KUKA KRL program: EPS_2_251806_MH50A_A_20260212042250.src

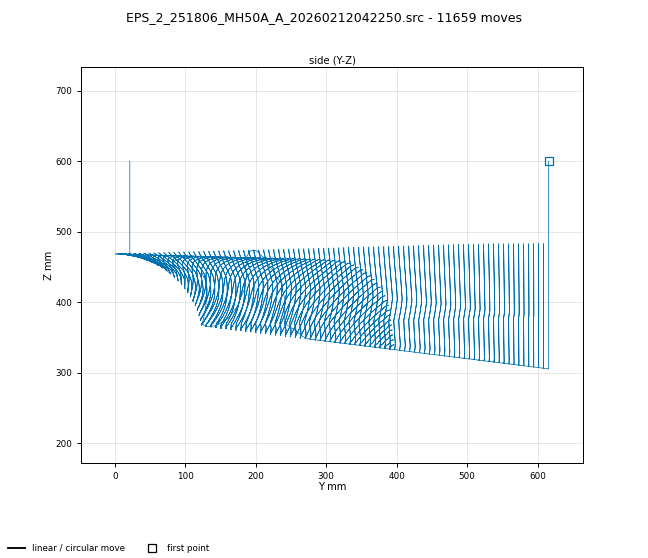
[picture p0: tool path of EPS_2_251806_MH50A_A_20260212042250.src, 11659 of 11661 moves have a stored position in this frame; points joined in program order, loops and branches not executed]
&ACCESS RVP
&REL 4
&COMMENT QRS 19112012
&PARAM EDITMASK = *
DEF PART()
EXT BAS (BAS_COMMAND :IN,REAL :IN )
INT I
BAS (#INITMOV,0 )

;KUKA QRS Post kuka4.cps  Date:22-06-2017 !

File_ID=3022

QRS_PRE_INIT()

;Init var - Until changes are made in qrs_pre_init
Outlet_Square_prg=0
Inlet_1_Square_prg=0
Inlet_2_Square_prg=0
Inlet_3_Square_prg=0
Inlet_4_Square_prg=0
Inlet_5_Square_prg=0

Outlet_1={X 0.000, Y 526.370, Z 382.500, B 0.000, E1 0.000 }
Inlet_1={X 0.000, Y 554.650, Z 357.500, B 0.000, E1 180.000 }
Outlet_1_type=201
Inlet_1_type=0
;QRS#1=Sidecore dimensions
;QRS#2=200-8" PVC SDR 35
;QRS#3=DeadEnd 201
;QRS#4=
;QRS#5=
;QRS#6=
;QRS#7=
;QRS#8=
;QRS#9=12-08 PSX
;QRS#10=

;QRS#11=
;QRS#12=
;QRS#13=
;QRS#14=
;QRS#15=
;QRS#16=1220x127x762 2,5'
;QRS#17=EPS Height
;QRS#18=483
;QRS#19=*
;QRS#20= UPDATED VERSION 22-06-2017
;QRS#21=*
Outlet_Square=0100
Inlet_1_Square=00
Inlet_2_Square=0
Inlet_3_Square=0
Inlet_4_Square=0
Inlet_5_Square=0
Mill_Square=1
Outlet_Square_Prg=204
Inlet_1_Square_prg=0

QRS_INIT()

$ADVANCE=5

; T1
PTP {E1 173.619,E2 173.619}
PTP {X 0,Y 615.481,A -85,B 0,C 180,E1 173.619,E2 173.619,E3 0,E4 0,E5 0,E6 0}
QRS_SPEED_INIT()
LIN {X 0,Y 615.481,Z 600,A -85,B 0,C 180,E1 173.619,E2 173.619,E3 0,E4 0,E5 0,E6 0} C_VEL
LIN {X 0,Y 615.481,Z 315.368,A -85,B 0,C 180,E1 173.619,E2 173.619} C_VEL
LIN {X 0,Y 615.481,Z 307.193,A -85,B 0,C 180,E1 173.619,E2 173.619} C_VEL
LIN {X 0,Y 615.471,Z 305.193,A -85,B 0,C 180,E1 173.433,E2 173.433} C_VEL
LIN {X 0,Y 615.484,Z 305.195,A -85,B 0,C 180,E1 170.802,E2 170.802} C_VEL
LIN {X 0,Y 615.484,Z 305.183,A -85,B 0,C 180,E1 168.14,E2 168.14} C_VEL
LIN {X 0,Y 615.479,Z 305.195,A -85,B 0,C 180,E1 165.451,E2 165.451} C_VEL
LIN {X 0,Y 615.484,Z 305.188,A -85,B 0,C 180,E1 162.73,E2 162.73} C_VEL
LIN {X 0,Y 615.472,Z 305.189,A -85,B 0,C 180,E1 159.967,E2 159.967} C_VEL
LIN {X 0,Y 615.478,Z 305.195,A -85,B 0,C 180,E1 157.656,E2 157.656} C_VEL
LIN {X 0,Y 615.483,Z 305.191,A -85,B 0,C 180,E1 155.009,E2 155.009} C_VEL
LIN {X 0,Y 615.486,Z 305.186,A -85,B 0,C 180,E1 152.823,E2 152.823} C_VEL
LIN {X 0,Y 615.473,Z 305.188,A -85,B 0,C 180,E1 150.207,E2 150.207} C_VEL
LIN {X 0,Y 615.495,Z 305.199,A -85,B 0,C 180,E1 147.544,E2 147.544} C_VEL
LIN {X 0,Y 615.482,Z 305.189,A -85,B 0,C 180,E1 145.185,E2 145.185} C_VEL
LIN {X 0,Y 615.492,Z 305.182,A -85,B 0,C 180,E1 142.759,E2 142.759} C_VEL
LIN {X 0,Y 615.49,Z 305.198,A -85,B 0,C 180,E1 139.91,E2 139.91} C_VEL
LIN {X 0,Y 615.488,Z 305.183,A -85,B 0,C 180,E1 136.952,E2 136.952} C_VEL
LIN {X 0,Y 615.483,Z 305.196,A -85,B 0,C 180,E1 134.15,E2 134.15} C_VEL
LIN {X 0,Y 615.482,Z 305.189,A -85,B 0,C 180,E1 131.474,E2 131.474} C_VEL
LIN {X 0,Y 615.483,Z 305.184,A -85,B 0,C 180,E1 128.904,E2 128.904} C_VEL
LIN {X 0,Y 615.479,Z 305.194,A -85,B 0,C 180,E1 126.425,E2 126.425} C_VEL
LIN {X 0,Y 615.484,Z 305.186,A -85,B 0,C 180,E1 123.534,E2 123.534} C_VEL
LIN {X 0,Y 615.477,Z 305.187,A -85,B 0,C 180,E1 120.92,E2 120.92} C_VEL
LIN {X 0,Y 615.489,Z 305.197,A -85,B 0,C 180,E1 118.451,E2 118.451} C_VEL
LIN {X 0,Y 615.486,Z 305.184,A -85,B 0,C 180,E1 115.57,E2 115.57} C_VEL
LIN {X 0,Y 615.475,Z 305.193,A -85,B 0,C 180,E1 112.845,E2 112.845} C_VEL
LIN {X 0,Y 615.491,Z 305.2,A -85,B 0,C 180,E1 110.559,E2 110.559} C_VEL
LIN {X 0,Y 615.48,Z 305.188,A -85,B 0,C 180,E1 107.957,E2 107.957} C_VEL
LIN {X 0,Y 615.477,Z 305.188,A -85,B 0,C 180,E1 105.226,E2 105.226} C_VEL
LIN {X 0,Y 615.488,Z 305.197,A -85,B 0,C 180,E1 102.53,E2 102.53} C_VEL
LIN {X 0,Y 615.494,Z 305.182,A -85,B 0,C 180,E1 99.862,E2 99.862} C_VEL
LIN {X 0,Y 615.475,Z 305.193,A -85,B 0,C 180,E1 97.216,E2 97.216} C_VEL
LIN {X 0,Y 615.481,Z 305.194,A -85,B 0,C 180,E1 94.585,E2 94.585} C_VEL
LIN {X 0,Y 615.5,Z 305.18,A -85,B 0,C 180,E1 91.963,E2 91.963} C_VEL
LIN {X 0,Y 615.48,Z 305.193,A -85,B 0,C 180,E1 89.346,E2 89.346} C_VEL
LIN {X 0,Y 615.48,Z 305.193,A -85,B 0,C 180,E1 86.727,E2 86.727} C_VEL
LIN {X 0,Y 615.498,Z 305.18,A -85,B 0,C 180,E1 84.102,E2 84.102} C_VEL
LIN {X 0,Y 615.484,Z 305.195,A -85,B 0,C 180,E1 81.463,E2 81.463} C_VEL
LIN {X 0,Y 615.477,Z 305.191,A -85,B 0,C 180,E1 78.807,E2 78.807} C_VEL
LIN {X 0,Y 615.484,Z 305.185,A -85,B 0,C 180,E1 76.067,E2 76.067} C_VEL
LIN {X 0,Y 615.49,Z 305.202,A -85,B 0,C 180,E1 73.414,E2 73.414} C_VEL
LIN {X 0,Y 615.483,Z 305.184,A -85,B 0,C 180,E1 70.662,E2 70.662} C_VEL
LIN {X 0,Y 615.482,Z 305.193,A -85,B 0,C 180,E1 67.863,E2 67.863} C_VEL
LIN {X 0,Y 615.475,Z 305.189,A -85,B 0,C 180,E1 65.008,E2 65.008} C_VEL
LIN {X 0,Y 615.482,Z 305.185,A -85,B 0,C 180,E1 62.823,E2 62.823} C_VEL
LIN {X 0,Y 615.48,Z 305.19,A -85,B 0,C 180,E1 60.206,E2 60.206} C_VEL
LIN {X 0,Y 615.482,Z 305.196,A -85,B 0,C 180,E1 57.542,E2 57.542} C_VEL
LIN {X 0,Y 615.476,Z 305.188,A -85,B 0,C 180,E1 55.184,E2 55.184} C_VEL
LIN {X 0,Y 615.493,Z 305.182,A -85,B 0,C 180,E1 52.758,E2 52.758} C_VEL
LIN {X 0,Y 615.495,Z 305.199,A -85,B 0,C 180,E1 49.91,E2 49.91} C_VEL
LIN {X 0,Y 615.488,Z 305.183,A -85,B 0,C 180,E1 46.952,E2 46.952} C_VEL
LIN {X 0,Y 615.49,Z 305.198,A -85,B 0,C 180,E1 43.998,E2 43.998} C_VEL
LIN {X 0,Y 615.487,Z 305.183,A -85,B 0,C 180,E1 41.095,E2 41.095} C_VEL
LIN {X 0,Y 615.485,Z 305.197,A -85,B 0,C 180,E1 38.068,E2 38.068} C_VEL
LIN {X 0,Y 615.471,Z 305.188,A -85,B 0,C 180,E1 35.616,E2 35.616} C_VEL
LIN {X 0,Y 615.487,Z 305.183,A -85,B 0,C 180,E1 33.236,E2 33.236} C_VEL
LIN {X 0,Y 615.483,Z 305.189,A -85,B 0,C 180,E1 30.919,E2 30.919} C_VEL
LIN {X 0,Y 615.493,Z 305.2,A -85,B 0,C 180,E1 28.452,E2 28.452} C_VEL
LIN {X 0,Y 615.484,Z 305.184,A -85,B 0,C 180,E1 25.569,E2 25.569} C_VEL
LIN {X 0,Y 615.484,Z 305.196,A -85,B 0,C 180,E1 22.844,E2 22.844} C_VEL
LIN {X 0,Y 615.483,Z 305.199,A -85,B 0,C 180,E1 20.557,E2 20.557} C_VEL
LIN {X 0,Y 615.475,Z 305.187,A -85,B 0,C 180,E1 17.957,E2 17.957} C_VEL
LIN {X 0,Y 615.482,Z 305.191,A -85,B 0,C 180,E1 15.226,E2 15.226} C_VEL
LIN {X 0,Y 615.475,Z 305.194,A -85,B 0,C 180,E1 12.53,E2 12.53} C_VEL
LIN {X 0,Y 615.492,Z 305.182,A -85,B 0,C 180,E1 9.862,E2 9.862} C_VEL
LIN {X 0,Y 615.488,Z 305.195,A -85,B 0,C 180,E1 7.215,E2 7.215} C_VEL
LIN {X 0,Y 615.471,Z 305.192,A -85,B 0,C 180,E1 4.584,E2 4.584} C_VEL
LIN {X 0,Y 615.5,Z 305.181,A -85,B 0,C 180,E1 1.963,E2 1.963} C_VEL
LIN {X 0,Y 615.491,Z 305.197,A -85,B 0,C 180,E1 -0.655,E2 -0.655} C_VEL
LIN {X 0,Y 615.469,Z 305.191,A -85,B 0,C 180,E1 -3.273,E2 -3.273} C_VEL
LIN {X 0,Y 615.498,Z 305.181,A -85,B 0,C 180,E1 -5.899,E2 -5.899} C_VEL
LIN {X 0,Y 615.494,Z 305.199,A -85,B 0,C 180,E1 -8.537,E2 -8.537} C_VEL
LIN {X 0,Y 615.468,Z 305.19,A -85,B 0,C 180,E1 -11.194,E2 -11.194} C_VEL
LIN {X 0,Y 615.488,Z 305.187,A -85,B 0,C 180,E1 -13.934,E2 -13.934} C_VEL
LIN {X 0,Y 615.481,Z 305.198,A -85,B 0,C 180,E1 -16.587,E2 -16.587} C_VEL
LIN {X 0,Y 615.48,Z 305.184,A -85,B 0,C 180,E1 -19.339,E2 -19.339} C_VEL
LIN {X 0,Y 615.488,Z 305.197,A -85,B 0,C 180,E1 -22.137,E2 -22.137} C_VEL
LIN {X 0,Y 615.469,Z 305.188,A -85,B 0,C 180,E1 -24.993,E2 -24.993} C_VEL
LIN {X 0,Y 615.489,Z 305.194,A -85,B 0,C 180,E1 -27.915,E2 -27.915} C_VEL
LIN {X 0,Y 615.491,Z 305.2,A -85,B 0,C 180,E1 -30.16,E2 -30.16} C_VEL
LIN {X 0,Y 615.469,Z 305.194,A -85,B 0,C 180,E1 -32.459,E2 -32.459} C_VEL
LIN {X 0,Y 615.47,Z 305.187,A -85,B 0,C 180,E1 -34.817,E2 -34.817} C_VEL
LIN {X 0,Y 615.494,Z 305.183,A -85,B 0,C 180,E1 -37.242,E2 -37.242} C_VEL
LIN {X 0,Y 615.479,Z 305.197,A -85,B 0,C 180,E1 -40.088,E2 -40.088} C_VEL
LIN {X 0,Y 615.465,Z 305.192,A -85,B 0,C 180,E1 -42.355,E2 -42.355} C_VEL
LIN {X 0,Y 615.491,Z 305.184,A -85,B 0,C 180,E1 -45.069,E2 -45.069} C_VEL
LIN {X 0,Y 615.488,Z 305.184,A -85,B 0,C 180,E1 -46.953,E2 -46.953} C_VEL
LIN {X 0,Y 615.499,Z 305.472,A -85,B 0,C 180,E1 -47.648,E2 -47.648} C_VEL
LIN {X 0,Y 615.458,Z 310.077,A -85,B 0,C 180,E1 -50.248,E2 -50.248} C_VEL
LIN {X 0,Y 615.486,Z 315.447,A -85,B 0,C 180,E1 -53.064,E2 -53.064} C_VEL
LIN {X 0,Y 615.483,Z 319.999,A -85,B 0,C 180,E1 -55.3,E2 -55.3} C_VEL
LIN {X 0,Y 615.457,Z 325.099,A -85,B 0,C 180,E1 -57.674,E2 -57.674} C_VEL
LIN {X 0,Y 615.477,Z 330.882,A -85,B 0,C 180,E1 -60.208,E2 -60.208} C_VEL
LIN {X 0,Y 615.484,Z 337.498,A -85,B 0,C 180,E1 -62.956,E2 -62.956} C_VEL
LIN {X 0,Y 615.466,Z 344.318,A -85,B 0,C 180,E1 -65.727,E2 -65.727} C_VEL
LIN {X 0,Y 615.496,Z 351.474,A -85,B 0,C 180,E1 -68.569,E2 -68.569} C_VEL
LIN {X 0,Y 615.462,Z 358.741,A -85,B 0,C 180,E1 -71.403,E2 -71.403} C_VEL
LIN {X 0,Y 615.472,Z 365.762,A -85,B 0,C 180,E1 -74.094,E2 -74.094} C_VEL
LIN {X 0,Y 615.482,Z 372.89,A -85,B 0,C 180,E1 -76.799,E2 -76.799} C_VEL
LIN {X 0,Y 615.496,Z 377.073,A -85,B 0,C 180,E1 -78.369,E2 -78.369} C_VEL
LIN {X 0,Y 615.477,Z 392.864,A -85,B 0,C 180,E1 -78.723,E2 -78.723} C_VEL
LIN {X 0,Y 615.442,Z 405.251,A -85,B 0,C 180,E1 -79.135,E2 -79.135} C_VEL
LIN {X 0,Y 615.442,Z 416.485,A -85,B 0,C 180,E1 -79.639,E2 -79.639} C_VEL
LIN {X 0,Y 615.493,Z 427.995,A -85,B 0,C 180,E1 -80.304,E2 -80.304} C_VEL
LIN {X 0,Y 615.499,Z 438.341,A -85,B 0,C 180,E1 -81.05,E2 -81.05} C_VEL
LIN {X 0,Y 615.497,Z 446.812,A -85,B 0,C 180,E1 -81.794,E2 -81.794} C_VEL
LIN {X 0,Y 615.498,Z 454.606,A -85,B 0,C 180,E1 -82.62,E2 -82.62} C_VEL
LIN {X 0,Y 615.496,Z 462.203,A -85,B 0,C 180,E1 -83.608,E2 -83.608} C_VEL
LIN {X 0,Y 615.498,Z 469.205,A -85,B 0,C 180,E1 -84.759,E2 -84.759} C_VEL
LIN {X 0,Y 615.494,Z 473.851,A -85,B 0,C 180,E1 -85.744,E2 -85.744} C_VEL
LIN {X 0,Y 615.494,Z 477.399,A -85,B 0,C 180,E1 -86.727,E2 -86.727} C_VEL
LIN {X 0,Y 615.497,Z 479.233,A -85,B 0,C 180,E1 -87.382,E2 -87.382} C_VEL
LIN {X 0,Y 615.5,Z 480.607,A -85,B 0,C 180,E1 -88.037,E2 -88.037} C_VEL
LIN {X 0,Y 615.496,Z 482.173,A -85,B 0,C 180,E1 -89.346,E2 -89.346} C_VEL
LIN {X 0,Y 615.494,Z 482.389,A -85,B 0,C 180,E1 -90,E2 -90} C_VEL
LIN {X 0,Y 615.495,Z 481.58,A -85,B 0,C 180,E1 -91.309,E2 -91.309} C_VEL
LIN {X 0,Y 615.5,Z 480.607,A -85,B 0,C 180,E1 -91.963,E2 -91.963} C_VEL
LIN {X 0,Y 615.497,Z 479.233,A -85,B 0,C 180,E1 -92.618,E2 -92.618} C_VEL
LIN {X 0,Y 615.496,Z 476.349,A -85,B 0,C 180,E1 -93.601,E2 -93.601} C_VEL
LIN {X 0,Y 615.498,Z 472.441,A -85,B 0,C 180,E1 -94.584,E2 -94.584} C_VEL
LIN {X 0,Y 615.499,Z 467.405,A -85,B 0,C 180,E1 -95.57,E2 -95.57} C_VEL
LIN {X 0,Y 615.497,Z 460.87,A -85,B 0,C 180,E1 -96.583,E2 -96.583} C_VEL
LIN {X 0,Y 615.497,Z 453.133,A -85,B 0,C 180,E1 -97.545,E2 -97.545} C_VEL
LIN {X 0,Y 615.498,Z 445.045,A -85,B 0,C 180,E1 -98.371,E2 -98.371} C_VEL
LIN {X 0,Y 615.499,Z 435.168,A -85,B 0,C 180,E1 -99.199,E2 -99.199} C_VEL
LIN {X 0,Y 615.478,Z 423.984,A -85,B 0,C 180,E1 -99.945,E2 -99.945} C_VEL
LIN {X 0,Y 615.436,Z 413.032,A -85,B 0,C 180,E1 -100.528,E2 -100.528} C_VEL
LIN {X 0,Y 615.452,Z 400.823,A -85,B 0,C 180,E1 -101.029,E2 -101.029} C_VEL
LIN {X 0,Y 615.49,Z 388.067,A -85,B 0,C 180,E1 -101.401,E2 -101.401} C_VEL
LIN {X 0,Y 615.496,Z 377.073,A -85,B 0,C 180,E1 -101.631,E2 -101.631} C_VEL
LIN {X 0,Y 615.472,Z 370.983,A -85,B 0,C 180,E1 -103.926,E2 -103.926} C_VEL
LIN {X 0,Y 615.454,Z 363.97,A -85,B 0,C 180,E1 -106.587,E2 -106.587} C_VEL
LIN {X 0,Y 615.493,Z 356.829,A -85,B 0,C 180,E1 -109.338,E2 -109.338} C_VEL
LIN {X 0,Y 615.463,Z 349.681,A -85,B 0,C 180,E1 -112.137,E2 -112.137} C_VEL
LIN {X 0,Y 615.487,Z 342.534,A -85,B 0,C 180,E1 -114.992,E2 -114.992} C_VEL
LIN {X 0,Y 615.486,Z 337.172,A -85,B 0,C 180,E1 -117.177,E2 -117.177} C_VEL
LIN {X 0,Y 615.477,Z 330.882,A -85,B 0,C 180,E1 -119.792,E2 -119.792} C_VEL
LIN {X 0,Y 615.457,Z 325.099,A -85,B 0,C 180,E1 -122.326,E2 -122.326} C_VEL
LIN {X 0,Y 615.496,Z 319.757,A -85,B 0,C 180,E1 -124.814,E2 -124.814} C_VEL
LIN {X 0,Y 615.495,Z 314.843,A -85,B 0,C 180,E1 -127.241,E2 -127.241} C_VEL
LIN {X 0,Y 615.458,Z 310.077,A -85,B 0,C 180,E1 -129.752,E2 -129.752} C_VEL
LIN {X 0,Y 615.499,Z 305.472,A -85,B 0,C 180,E1 -132.352,E2 -132.352} C_VEL
LIN {X 0,Y 615.486,Z 305.198,A -85,B 0,C 180,E1 -134.149,E2 -134.149} C_VEL
LIN {X 0,Y 615.488,Z 305.184,A -85,B 0,C 180,E1 -136.952,E2 -136.952} C_VEL
LIN {X 0,Y 615.467,Z 305.189,A -85,B 0,C 180,E1 -139.392,E2 -139.392} C_VEL
LIN {X 0,Y 615.48,Z 305.2,A -85,B 0,C 180,E1 -141.989,E2 -141.989} C_VEL
LIN {X 0,Y 615.484,Z 305.192,A -85,B 0,C 180,E1 -144.384,E2 -144.384} C_VEL
LIN {X 0,Y 615.487,Z 305.184,A -85,B 0,C 180,E1 -146.763,E2 -146.763} C_VEL
LIN {X 0,Y 615.47,Z 305.187,A -85,B 0,C 180,E1 -149.079,E2 -149.079} C_VEL
LIN {X 0,Y 615.474,Z 305.195,A -85,B 0,C 180,E1 -151.552,E2 -151.552} C_VEL
LIN {X 0,Y 615.488,Z 305.185,A -85,B 0,C 180,E1 -154.431,E2 -154.431} C_VEL
LIN {X 0,Y 615.467,Z 305.191,A -85,B 0,C 180,E1 -157.154,E2 -157.154} C_VEL
LIN {X 0,Y 615.48,Z 305.196,A -85,B 0,C 180,E1 -159.444,E2 -159.444} C_VEL
LIN {X 0,Y 615.486,Z 305.19,A -85,B 0,C 180,E1 -162.043,E2 -162.043} C_VEL
LIN {X 0,Y 615.47,Z 305.188,A -85,B 0,C 180,E1 -164.773,E2 -164.773} C_VEL
LIN {X 0,Y 615.487,Z 305.203,A -85,B 0,C 180,E1 -167.47,E2 -167.47} C_VEL
LIN {X 0,Y 615.495,Z 305.183,A -85,B 0,C 180,E1 -170.138,E2 -170.138} C_VEL
LIN {X 0,Y 615.469,Z 305.191,A -85,B 0,C 180,E1 -172.784,E2 -172.784} C_VEL
LIN {X 0,Y 615.492,Z 305.197,A -85,B 0,C 180,E1 -175.415,E2 -175.415} C_VEL
LIN {X 0,Y 615.5,Z 305.181,A -85,B 0,C 180,E1 -178.037,E2 -178.037} C_VEL
LIN {X 0,Y 615.47,Z 305.192,A -85,B 0,C 180,E1 -180.654,E2 -180.654} C_VEL
LIN {X 0,Y 615.49,Z 305.196,A -85,B 0,C 180,E1 -183.273,E2 -183.273} C_VEL
LIN {X 0,Y 615.497,Z 305.181,A -85,B 0,C 180,E1 -185.898,E2 -185.898} C_VEL
LIN {X 0,Y 615.471,Z 305.193,A -85,B 0,C 180,E1 -186.567,E2 -186.567} C_VEL
LIN {X 0,Y 614.806,Z 305.344,A -85,B 0,C 180,E1 -187.113,E2 -187.113} C_VEL
LIN {X 0,Y 611.977,Z 305.748,A -85,B 0,C 180,E1 -187.999,E2 -187.999} C_VEL
LIN {X 0,Y 609.585,Z 306.062,A -85,B 0,C 180,E1 -188.712,E2 -188.712} C_VEL
LIN {X 0,Y 608.549,Z 306.181,A -85,B 0,C 180,E1 -189.262,E2 -189.262} C_VEL
LIN {X 0,Y 608.46,Z 306.189,A -85,B 0,C 180,E1 -189.448,E2 -189.448} C_VEL
LIN {X 0,Y 608.458,Z 306.187,A -85,B 0,C 180,E1 -191.999,E2 -191.999} C_VEL
LIN {X 0,Y 608.469,Z 306.194,A -85,B 0,C 180,E1 -194.72,E2 -194.72} C_VEL
LIN {X 0,Y 608.448,Z 306.189,A -85,B 0,C 180,E1 -197.476,E2 -197.476} C_VEL
LIN {X 0,Y 608.454,Z 306.191,A -85,B 0,C 180,E1 -200.274,E2 -200.274} C_VEL
LIN {X 0,Y 608.456,Z 306.195,A -85,B 0,C 180,E1 -202.476,E2 -202.476} C_VEL
LIN {X 0,Y 608.45,Z 306.189,A -85,B 0,C 180,E1 -205.301,E2 -205.301} C_VEL
LIN {X 0,Y 608.444,Z 306.189,A -85,B 0,C 180,E1 -207.518,E2 -207.518} C_VEL
LIN {X 0,Y 608.456,Z 306.19,A -85,B 0,C 180,E1 -209.97,E2 -209.97} C_VEL
LIN {X 0,Y 608.468,Z 306.194,A -85,B 0,C 180,E1 -212.524,E2 -212.524} C_VEL
LIN {X 0,Y 608.435,Z 306.19,A -85,B 0,C 180,E1 -215.278,E2 -215.278} C_VEL
LIN {X 0,Y 608.468,Z 306.188,A -85,B 0,C 180,E1 -217.746,E2 -217.746} C_VEL
LIN {X 0,Y 608.452,Z 306.196,A -85,B 0,C 180,E1 -220.329,E2 -220.329} C_VEL
LIN {X 0,Y 608.454,Z 306.188,A -85,B 0,C 180,E1 -222.959,E2 -222.959} C_VEL
LIN {X 0,Y 608.454,Z 306.192,A -85,B 0,C 180,E1 -225.736,E2 -225.736} C_VEL
LIN {X 0,Y 608.46,Z 306.188,A -85,B 0,C 180,E1 -228.657,E2 -228.657} C_VEL
LIN {X 0,Y 608.467,Z 306.188,A -85,B 0,C 180,E1 -231.412,E2 -231.412} C_VEL
LIN {X 0,Y 608.473,Z 306.194,A -85,B 0,C 180,E1 -233.95,E2 -233.95} C_VEL
LIN {X 0,Y 608.463,Z 306.189,A -85,B 0,C 180,E1 -236.329,E2 -236.329} C_VEL
LIN {X 0,Y 608.474,Z 306.185,A -85,B 0,C 180,E1 -238.727,E2 -238.727} C_VEL
LIN {X 0,Y 608.47,Z 306.19,A -85,B 0,C 180,E1 -241.38,E2 -241.38} C_VEL
LIN {X 0,Y 608.469,Z 306.187,A -85,B 0,C 180,E1 -244.279,E2 -244.279} C_VEL
LIN {X 0,Y 608.445,Z 306.19,A -85,B 0,C 180,E1 -246.876,E2 -246.876} C_VEL
LIN {X 0,Y 608.467,Z 306.193,A -85,B 0,C 180,E1 -249.32,E2 -249.32} C_VEL
LIN {X 0,Y 608.448,Z 306.192,A -85,B 0,C 180,E1 -251.828,E2 -251.828} C_VEL
LIN {X 0,Y 608.464,Z 306.187,A -85,B 0,C 180,E1 -254.594,E2 -254.594} C_VEL
LIN {X 0,Y 608.474,Z 306.195,A -85,B 0,C 180,E1 -257.323,E2 -257.323} C_VEL
LIN {X 0,Y 608.461,Z 306.187,A -85,B 0,C 180,E1 -260.023,E2 -260.023} C_VEL
LIN {X 0,Y 608.456,Z 306.19,A -85,B 0,C 180,E1 -262.701,E2 -262.701} C_VEL
LIN {X 0,Y 608.46,Z 306.19,A -85,B 0,C 180,E1 -264.698,E2 -264.698} C_VEL
LIN {X 0,Y 608.472,Z 306.191,A -85,B 0,C 180,E1 -267.352,E2 -267.352} C_VEL
LIN {X 0,Y 608.477,Z 306.185,A -85,B 0,C 180,E1 -270,E2 -270} C_VEL
LIN {X 0,Y 608.472,Z 306.191,A -85,B 0,C 180,E1 -272.648,E2 -272.648} C_VEL
LIN {X 0,Y 608.46,Z 306.19,A -85,B 0,C 180,E1 -275.302,E2 -275.302} C_VEL
LIN {X 0,Y 608.477,Z 306.185,A -85,B 0,C 180,E1 -277.967,E2 -277.967} C_VEL
LIN {X 0,Y 608.468,Z 306.192,A -85,B 0,C 180,E1 -280.958,E2 -280.958} C_VEL
LIN {X 0,Y 608.457,Z 306.188,A -85,B 0,C 180,E1 -283.357,E2 -283.357} C_VEL
LIN {X 0,Y 608.458,Z 306.189,A -85,B 0,C 180,E1 -286.094,E2 -286.094} C_VEL
LIN {X 0,Y 608.457,Z 306.192,A -85,B 0,C 180,E1 -288.869,E2 -288.869} C_VEL
LIN {X 0,Y 608.47,Z 306.186,A -85,B 0,C 180,E1 -291.691,E2 -291.691} C_VEL
LIN {X 0,Y 608.45,Z 306.195,A -85,B 0,C 180,E1 -294.571,E2 -294.571} C_VEL
LIN {X 0,Y 608.474,Z 306.185,A -85,B 0,C 180,E1 -297.207,E2 -297.207} C_VEL
LIN {X 0,Y 608.465,Z 306.191,A -85,B 0,C 180,E1 -299.972,E2 -299.972} C_VEL
LIN {X 0,Y 608.458,Z 306.192,A -85,B 0,C 180,E1 -302.523,E2 -302.523} C_VEL
LIN {X 0,Y 608.436,Z 306.19,A -85,B 0,C 180,E1 -305.278,E2 -305.278} C_VEL
LIN {X 0,Y 608.471,Z 306.19,A -85,B 0,C 180,E1 -307.746,E2 -307.746} C_VEL
LIN {X 0,Y 608.45,Z 306.193,A -85,B 0,C 180,E1 -310.33,E2 -310.33} C_VEL
LIN {X 0,Y 608.453,Z 306.187,A -85,B 0,C 180,E1 -312.96,E2 -312.96} C_VEL
LIN {X 0,Y 608.464,Z 306.194,A -85,B 0,C 180,E1 -315.735,E2 -315.735} C_VEL
LIN {X 0,Y 608.457,Z 306.187,A -85,B 0,C 180,E1 -318.658,E2 -318.658} C_VEL
LIN {X 0,Y 608.468,Z 306.19,A -85,B 0,C 180,E1 -321.413,E2 -321.413} C_VEL
LIN {X 0,Y 608.442,Z 306.195,A -85,B 0,C 180,E1 -323.955,E2 -323.955} C_VEL
LIN {X 0,Y 608.446,Z 306.189,A -85,B 0,C 180,E1 -326.329,E2 -326.329} C_VEL
LIN {X 0,Y 608.475,Z 306.185,A -85,B 0,C 180,E1 -328.728,E2 -328.728} C_VEL
LIN {X 0,Y 608.475,Z 306.193,A -85,B 0,C 180,E1 -331.379,E2 -331.379} C_VEL
LIN {X 0,Y 608.441,Z 306.191,A -85,B 0,C 180,E1 -333.965,E2 -333.965} C_VEL
LIN {X 0,Y 608.457,Z 306.188,A -85,B 0,C 180,E1 -336.155,E2 -336.155} C_VEL
LIN {X 0,Y 608.468,Z 306.186,A -85,B 0,C 180,E1 -338.309,E2 -338.309} C_VEL
LIN {X 0,Y 608.469,Z 306.196,A -85,B 0,C 180,E1 -341.284,E2 -341.284} C_VEL
LIN {X 0,Y 608.453,Z 306.188,A -85,B 0,C 180,E1 -343.906,E2 -343.906} C_VEL
LIN {X 0,Y 608.462,Z 306.189,A -85,B 0,C 180,E1 -346.644,E2 -346.644} C_VEL
LIN {X 0,Y 608.457,Z 306.193,A -85,B 0,C 180,E1 -349.35,E2 -349.35} C_VEL
LIN {X 0,Y 608.475,Z 306.185,A -85,B 0,C 180,E1 -352.033,E2 -352.033} C_VEL
LIN {X 0,Y 608.468,Z 306.192,A -85,B 0,C 180,E1 -354.699,E2 -354.699} C_VEL
LIN {X 0,Y 608.463,Z 306.189,A -85,B 0,C 180,E1 -357.352,E2 -357.352} C_VEL
LIN {X 0,Y 608.477,Z 306.185,A -85,B 0,C 180,E1 -360,E2 -360} C_VEL
LIN {X 0,Y 608.478,Z 306.193,A -85,B 0,C 180,E1 -362.648,E2 -362.648} C_VEL
LIN {X 0,Y 608.451,Z 306.189,A -85,B 0,C 180,E1 -365.302,E2 -365.302} C_VEL
LIN {X 0,Y 608.479,Z 306.185,A -85,B 0,C 180,E1 -367.967,E2 -367.967} C_VEL
LIN {X 0,Y 608.463,Z 306.19,A -85,B 0,C 180,E1 -370.954,E2 -370.954} C_VEL
LIN {X 0,Y 608.452,Z 306.188,A -85,B 0,C 180,E1 -373.357,E2 -373.357} C_VEL
LIN {X 0,Y 608.463,Z 306.191,A -85,B 0,C 180,E1 -376.094,E2 -376.094} C_VEL
LIN {X 0,Y 608.451,Z 306.19,A -85,B 0,C 180,E1 -378.87,E2 -378.87} C_VEL
LIN {X 0,Y 608.472,Z 306.187,A -85,B 0,C 180,E1 -381.692,E2 -381.692} C_VEL
LIN {X 0,Y 608.448,Z 306.193,A -85,B 0,C 180,E1 -384.572,E2 -384.572} C_VEL
LIN {X 0,Y 608.472,Z 306.185,A -85,B 0,C 180,E1 -387.206,E2 -387.206} C_VEL
LIN {X 0,Y 608.47,Z 306.194,A -85,B 0,C 180,E1 -389.972,E2 -389.972} C_VEL
LIN {X 0,Y 608.452,Z 306.188,A -85,B 0,C 180,E1 -392.88,E2 -392.88} C_VEL
LIN {X 0,Y 608.436,Z 306.191,A -85,B 0,C 180,E1 -395.278,E2 -395.278} C_VEL
LIN {X 0,Y 608.469,Z 306.193,A -85,B 0,C 180,E1 -397.747,E2 -397.747} C_VEL
LIN {X 0,Y 608.438,Z 306.192,A -85,B 0,C 180,E1 -400.328,E2 -400.328} C_VEL
LIN {X 0,Y 608.478,Z 306.188,A -85,B 0,C 180,E1 -403.31,E2 -403.31} C_VEL
LIN {X 0,Y 608.461,Z 306.191,A -85,B 0,C 180,E1 -406.13,E2 -406.13} C_VEL
LIN {X 0,Y 608.451,Z 306.19,A -85,B 0,C 180,E1 -407.04,E2 -407.04} C_VEL
LIN {X 0,Y 608.491,Z 307.285,A -85,B 0,C 180,E1 -407.941,E2 -407.941} C_VEL
LIN {X 0,Y 608.5,Z 312.161,A -85,B 0,C 180,E1 -410.7,E2 -410.7} C_VEL
LIN {X 0,Y 608.511,Z 316.701,A -85,B 0,C 180,E1 -413.089,E2 -413.089} C_VEL
LIN {X 0,Y 608.458,Z 321.649,A -85,B 0,C 180,E1 -415.53,E2 -415.53} C_VEL
LIN {X 0,Y 608.452,Z 326.723,A -85,B 0,C 180,E1 -417.905,E2 -417.905} C_VEL
LIN {X 0,Y 608.462,Z 331.937,A -85,B 0,C 180,E1 -420.22,E2 -420.22} C_VEL
LIN {X 0,Y 608.459,Z 338.084,A -85,B 0,C 180,E1 -422.797,E2 -422.797} C_VEL
LIN {X 0,Y 608.445,Z 344.512,A -85,B 0,C 180,E1 -425.429,E2 -425.429} C_VEL
LIN {X 0,Y 608.435,Z 349.902,A -85,B 0,C 180,E1 -427.593,E2 -427.593} C_VEL
LIN {X 0,Y 608.448,Z 357.088,A -85,B 0,C 180,E1 -430.429,E2 -430.429} C_VEL
LIN {X 0,Y 608.402,Z 364.274,A -85,B 0,C 180,E1 -433.215,E2 -433.215} C_VEL
LIN {X 0,Y 608.391,Z 369.664,A -85,B 0,C 180,E1 -435.278,E2 -435.278} C_VEL
LIN {X 0,Y 608.449,Z 377.299,A -85,B 0,C 180,E1 -438.169,E2 -438.169} C_VEL
LIN {X 0,Y 608.459,Z 377.616,A -85,B 0,C 180,E1 -438.254,E2 -438.254} C_VEL
LIN {X 0,Y 608.541,Z 390.705,A -85,B 0,C 180,E1 -438.53,E2 -438.53} C_VEL
LIN {X 0,Y 608.472,Z 403.565,A -85,B 0,C 180,E1 -438.941,E2 -438.941} C_VEL
LIN {X 0,Y 608.466,Z 414.924,A -85,B 0,C 180,E1 -439.434,E2 -439.434} C_VEL
LIN {X 0,Y 608.478,Z 425.579,A -85,B 0,C 180,E1 -440.023,E2 -440.023} C_VEL
LIN {X 0,Y 608.483,Z 436.476,A -85,B 0,C 180,E1 -440.778,E2 -440.778} C_VEL
LIN {X 0,Y 608.475,Z 447.114,A -85,B 0,C 180,E1 -441.699,E2 -441.699} C_VEL
LIN {X 0,Y 608.471,Z 454.96,A -85,B 0,C 180,E1 -442.534,E2 -442.534} C_VEL
LIN {X 0,Y 608.461,Z 462.286,A -85,B 0,C 180,E1 -443.485,E2 -443.485} C_VEL
LIN {X 0,Y 608.451,Z 467.865,A -85,B 0,C 180,E1 -444.366,E2 -444.366} C_VEL
LIN {X 0,Y 608.432,Z 472.95,A -85,B 0,C 180,E1 -445.362,E2 -445.362} C_VEL
LIN {X 0,Y 608.449,Z 476.896,A -85,B 0,C 180,E1 -446.358,E2 -446.358} C_VEL
LIN {X 0,Y 608.425,Z 479.808,A -85,B 0,C 180,E1 -447.352,E2 -447.352} C_VEL
LIN {X 0,Y 608.445,Z 481.201,A -85,B 0,C 180,E1 -448.014,E2 -448.014} C_VEL
LIN {X 0,Y 608.438,Z 482.783,A -85,B 0,C 180,E1 -449.338,E2 -449.338} C_VEL
LIN {X 0,Y 608.434,Z 482.998,A -85,B 0,C 180,E1 -450,E2 -450} C_VEL
LIN {X 0,Y 608.448,Z 482.184,A -85,B 0,C 180,E1 -451.324,E2 -451.324} C_VEL
LIN {X 0,Y 608.445,Z 481.201,A -85,B 0,C 180,E1 -451.986,E2 -451.986} C_VEL
LIN {X 0,Y 608.425,Z 479.808,A -85,B 0,C 180,E1 -452.648,E2 -452.648} C_VEL
LIN {X 0,Y 608.449,Z 476.896,A -85,B 0,C 180,E1 -453.642,E2 -453.642} C_VEL
LIN {X 0,Y 608.432,Z 472.95,A -85,B 0,C 180,E1 -454.638,E2 -454.638} C_VEL
LIN {X 0,Y 608.451,Z 467.865,A -85,B 0,C 180,E1 -455.634,E2 -455.634} C_VEL
LIN {X 0,Y 608.442,Z 461.472,A -85,B 0,C 180,E1 -456.633,E2 -456.633} C_VEL
LIN {X 0,Y 608.475,Z 453.479,A -85,B 0,C 180,E1 -457.633,E2 -457.633} C_VEL
LIN {X 0,Y 608.487,Z 445.338,A -85,B 0,C 180,E1 -458.468,E2 -458.468} C_VEL
LIN {X 0,Y 608.487,Z 435.398,A -85,B 0,C 180,E1 -459.306,E2 -459.306} C_VEL
LIN {X 0,Y 608.484,Z 424.168,A -85,B 0,C 180,E1 -460.061,E2 -460.061} C_VEL
LIN {X 0,Y 608.46,Z 411.891,A -85,B 0,C 180,E1 -460.712,E2 -460.712} C_VEL
LIN {X 0,Y 608.487,Z 400.098,A -85,B 0,C 180,E1 -461.186,E2 -461.186} C_VEL
LIN {X 0,Y 608.548,Z 387.262,A -85,B 0,C 180,E1 -461.554,E2 -461.554} C_VEL
LIN {X 0,Y 608.436,Z 377.467,A -85,B 0,C 180,E1 -461.768,E2 -461.768} C_VEL
LIN {X 0,Y 608.426,Z 371.46,A -85,B 0,C 180,E1 -464.038,E2 -464.038} C_VEL
LIN {X 0,Y 608.402,Z 364.274,A -85,B 0,C 180,E1 -466.785,E2 -466.785} C_VEL
LIN {X 0,Y 608.449,Z 357.088,A -85,B 0,C 180,E1 -469.571,E2 -469.571} C_VEL
LIN {X 0,Y 608.431,Z 349.746,A -85,B 0,C 180,E1 -472.469,E2 -472.469} C_VEL
LIN {X 0,Y 608.445,Z 344.512,A -85,B 0,C 180,E1 -474.571,E2 -474.571} C_VEL
LIN {X 0,Y 608.459,Z 338.084,A -85,B 0,C 180,E1 -477.203,E2 -477.203} C_VEL
LIN {X 0,Y 608.462,Z 331.489,A -85,B 0,C 180,E1 -479.97,E2 -479.97} C_VEL
LIN {X 0,Y 608.461,Z 325.787,A -85,B 0,C 180,E1 -482.522,E2 -482.522} C_VEL
LIN {X 0,Y 608.471,Z 319.985,A -85,B 0,C 180,E1 -485.276,E2 -485.276} C_VEL
LIN {X 0,Y 608.487,Z 315.09,A -85,B 0,C 180,E1 -487.745,E2 -487.745} C_VEL
LIN {X 0,Y 608.485,Z 310.293,A -85,B 0,C 180,E1 -490.332,E2 -490.332} C_VEL
LIN {X 0,Y 608.514,Z 306.802,A -85,B 0,C 180,E1 -492.339,E2 -492.339} C_VEL
LIN {X 0,Y 608.451,Z 306.191,A -85,B 0,C 180,E1 -492.96,E2 -492.96} C_VEL
LIN {X 0,Y 608.443,Z 306.192,A -85,B 0,C 180,E1 -495.737,E2 -495.737} C_VEL
LIN {X 0,Y 608.456,Z 306.193,A -85,B 0,C 180,E1 -497.938,E2 -497.938} C_VEL
LIN {X 0,Y 608.48,Z 306.186,A -85,B 0,C 180,E1 -500.701,E2 -500.701} C_VEL
LIN {X 0,Y 608.449,Z 306.188,A -85,B 0,C 180,E1 -503.084,E2 -503.084} C_VEL
LIN {X 0,Y 608.459,Z 306.19,A -85,B 0,C 180,E1 -505.53,E2 -505.53} C_VEL
LIN {X 0,Y 608.46,Z 306.196,A -85,B 0,C 180,E1 -507.905,E2 -507.905} C_VEL
LIN {X 0,Y 608.472,Z 306.19,A -85,B 0,C 180,E1 -510.22,E2 -510.22} C_VEL
LIN {X 0,Y 608.472,Z 306.185,A -85,B 0,C 180,E1 -512.794,E2 -512.794} C_VEL
LIN {X 0,Y 608.448,Z 306.193,A -85,B 0,C 180,E1 -515.428,E2 -515.428} C_VEL
LIN {X 0,Y 608.472,Z 306.187,A -85,B 0,C 180,E1 -518.308,E2 -518.308} C_VEL
LIN {X 0,Y 608.466,Z 306.19,A -85,B 0,C 180,E1 -521.285,E2 -521.285} C_VEL
LIN {X 0,Y 608.463,Z 306.191,A -85,B 0,C 180,E1 -523.906,E2 -523.906} C_VEL
LIN {X 0,Y 608.452,Z 306.188,A -85,B 0,C 180,E1 -526.643,E2 -526.643} C_VEL
LIN {X 0,Y 608.463,Z 306.195,A -85,B 0,C 180,E1 -529.35,E2 -529.35} C_VEL
LIN {X 0,Y 608.479,Z 306.185,A -85,B 0,C 180,E1 -532.033,E2 -532.033} C_VEL
LIN {X 0,Y 608.45,Z 306.189,A -85,B 0,C 180,E1 -534.698,E2 -534.698} C_VEL
LIN {X 0,Y 608.478,Z 306.193,A -85,B 0,C 180,E1 -537.352,E2 -537.352} C_VEL
LIN {X 0,Y 608.477,Z 306.185,A -85,B 0,C 180,E1 -540,E2 -540} C_VEL
LIN {X 0,Y 608.463,Z 306.189,A -85,B 0,C 180,E1 -542.648,E2 -542.648} C_VEL
LIN {X 0,Y 608.468,Z 306.192,A -85,B 0,C 180,E1 -545.301,E2 -545.301} C_VEL
LIN {X 0,Y 608.475,Z 306.185,A -85,B 0,C 180,E1 -547.967,E2 -547.967} C_VEL
LIN {X 0,Y 608.46,Z 306.189,A -85,B 0,C 180,E1 -549.448,E2 -549.448} C_VEL
LIN {X 0,Y 607.781,Z 306.274,A -85,B 0,C 180,E1 -550,E2 -550} C_VEL
LIN {X 0,Y 604.927,Z 306.637,A -85,B 0,C 180,E1 -550.897,E2 -550.897} C_VEL
LIN {X 0,Y 602.522,Z 306.931,A -85,B 0,C 180,E1 -551.619,E2 -551.619} C_VEL
LIN {X 0,Y 601.49,Z 307.056,A -85,B 0,C 180,E1 -552.175,E2 -552.175} C_VEL
LIN {X 0,Y 601.405,Z 307.068,A -85,B 0,C 180,E1 -552.364,E2 -552.364} C_VEL
LIN {X 0,Y 601.425,Z 307.072,A -85,B 0,C 180,E1 -554.897,E2 -554.897} C_VEL
LIN {X 0,Y 601.43,Z 307.069,A -85,B 0,C 180,E1 -556.986,E2 -556.986} C_VEL
LIN {X 0,Y 601.401,Z 307.066,A -85,B 0,C 180,E1 -559.809,E2 -559.809} C_VEL
LIN {X 0,Y 601.413,Z 307.075,A -85,B 0,C 180,E1 -562.605,E2 -562.605} C_VEL
LIN {X 0,Y 601.399,Z 307.071,A -85,B 0,C 180,E1 -564.878,E2 -564.878} C_VEL
LIN {X 0,Y 601.414,Z 307.065,A -85,B 0,C 180,E1 -567.363,E2 -567.363} C_VEL
LIN {X 0,Y 601.424,Z 307.068,A -85,B 0,C 180,E1 -570.148,E2 -570.148} C_VEL
LIN {X 0,Y 601.427,Z 307.068,A -85,B 0,C 180,E1 -572.717,E2 -572.717} C_VEL
LIN {X 0,Y 601.392,Z 307.068,A -85,B 0,C 180,E1 -575.112,E2 -575.112} C_VEL
LIN {X 0,Y 601.433,Z 307.062,A -85,B 0,C 180,E1 -577.419,E2 -577.419} C_VEL
LIN {X 0,Y 601.409,Z 307.072,A -85,B 0,C 180,E1 -579.995,E2 -579.995} C_VEL
LIN {X 0,Y 601.41,Z 307.067,A -85,B 0,C 180,E1 -582.67,E2 -582.67} C_VEL
LIN {X 0,Y 601.422,Z 307.065,A -85,B 0,C 180,E1 -585.482,E2 -585.482} C_VEL
LIN {X 0,Y 601.423,Z 307.067,A -85,B 0,C 180,E1 -588.406,E2 -588.406} C_VEL
LIN {X 0,Y 601.435,Z 307.062,A -85,B 0,C 180,E1 -590.876,E2 -590.876} C_VEL
LIN {X 0,Y 601.439,Z 307.069,A -85,B 0,C 180,E1 -593.734,E2 -593.734} C_VEL
LIN {X 0,Y 601.426,Z 307.063,A -85,B 0,C 180,E1 -596.687,E2 -596.687} C_VEL
LIN {X 0,Y 601.427,Z 307.064,A -85,B 0,C 180,E1 -599.059,E2 -599.059} C_VEL
LIN {X 0,Y 601.43,Z 307.067,A -85,B 0,C 180,E1 -601.373,E2 -601.373} C_VEL
LIN {X 0,Y 601.402,Z 307.077,A -85,B 0,C 180,E1 -603.636,E2 -603.636} C_VEL
LIN {X 0,Y 601.416,Z 307.064,A -85,B 0,C 180,E1 -606.59,E2 -606.59} C_VEL
LIN {X 0,Y 601.43,Z 307.073,A -85,B 0,C 180,E1 -609.478,E2 -609.478} C_VEL
LIN {X 0,Y 601.393,Z 307.067,A -85,B 0,C 180,E1 -612.312,E2 -612.312} C_VEL
LIN {X 0,Y 601.409,Z 307.065,A -85,B 0,C 180,E1 -614.409,E2 -614.409} C_VEL
LIN {X 0,Y 601.418,Z 307.072,A -85,B 0,C 180,E1 -617.172,E2 -617.172} C_VEL
LIN {X 0,Y 601.437,Z 307.063,A -85,B 0,C 180,E1 -619.905,E2 -619.905} C_VEL
LIN {X 0,Y 601.435,Z 307.064,A -85,B 0,C 180,E1 -622.615,E2 -622.615} C_VEL
LIN {X 0,Y 601.418,Z 307.071,A -85,B 0,C 180,E1 -625.308,E2 -625.308} C_VEL
LIN {X 0,Y 601.438,Z 307.062,A -85,B 0,C 180,E1 -627.991,E2 -627.991} C_VEL
LIN {X 0,Y 601.446,Z 307.066,A -85,B 0,C 180,E1 -630.67,E2 -630.67} C_VEL
LIN {X 0,Y 601.425,Z 307.067,A -85,B 0,C 180,E1 -633.35,E2 -633.35} C_VEL
LIN {X 0,Y 601.441,Z 307.062,A -85,B 0,C 180,E1 -636.037,E2 -636.037} C_VEL
LIN {X 0,Y 601.433,Z 307.072,A -85,B 0,C 180,E1 -638.738,E2 -638.738} C_VEL
LIN {X 0,Y 601.431,Z 307.063,A -85,B 0,C 180,E1 -641.458,E2 -641.458} C_VEL
LIN {X 0,Y 601.417,Z 307.068,A -85,B 0,C 180,E1 -644.205,E2 -644.205} C_VEL
LIN {X 0,Y 601.43,Z 307.067,A -85,B 0,C 180,E1 -646.986,E2 -646.986} C_VEL
LIN {X 0,Y 601.404,Z 307.067,A -85,B 0,C 180,E1 -649.809,E2 -649.809} C_VEL
LIN {X 0,Y 601.412,Z 307.072,A -85,B 0,C 180,E1 -652.606,E2 -652.606} C_VEL
LIN {X 0,Y 601.4,Z 307.069,A -85,B 0,C 180,E1 -654.879,E2 -654.879} C_VEL
LIN {X 0,Y 601.419,Z 307.067,A -85,B 0,C 180,E1 -657.867,E2 -657.867} C_VEL
LIN {X 0,Y 601.425,Z 307.072,A -85,B 0,C 180,E1 -660.164,E2 -660.164} C_VEL
LIN {X 0,Y 601.419,Z 307.066,A -85,B 0,C 180,E1 -662.716,E2 -662.716} C_VEL
LIN {X 0,Y 601.391,Z 307.067,A -85,B 0,C 180,E1 -665.112,E2 -665.112} C_VEL
LIN {X 0,Y 601.434,Z 307.063,A -85,B 0,C 180,E1 -667.419,E2 -667.419} C_VEL
LIN {X 0,Y 601.41,Z 307.075,A -85,B 0,C 180,E1 -669.995,E2 -669.995} C_VEL
LIN {X 0,Y 601.408,Z 307.066,A -85,B 0,C 180,E1 -672.67,E2 -672.67} C_VEL
LIN {X 0,Y 601.422,Z 307.067,A -85,B 0,C 180,E1 -675.482,E2 -675.482} C_VEL
LIN {X 0,Y 601.422,Z 307.065,A -85,B 0,C 180,E1 -678.407,E2 -678.407} C_VEL
LIN {X 0,Y 601.435,Z 307.062,A -85,B 0,C 180,E1 -680.876,E2 -680.876} C_VEL
LIN {X 0,Y 601.402,Z 307.071,A -85,B 0,C 180,E1 -683.418,E2 -683.418} C_VEL
LIN {X 0,Y 601.428,Z 307.066,A -85,B 0,C 180,E1 -686.065,E2 -686.065} C_VEL
LIN {X 0,Y 601.438,Z 307.061,A -85,B 0,C 180,E1 -688.542,E2 -688.542} C_VEL
LIN {X 0,Y 601.434,Z 307.07,A -85,B 0,C 180,E1 -691.374,E2 -691.374} C_VEL
LIN {X 0,Y 601.4,Z 307.073,A -85,B 0,C 180,E1 -693.637,E2 -693.637} C_VEL
LIN {X 0,Y 601.416,Z 307.065,A -85,B 0,C 180,E1 -696.59,E2 -696.59} C_VEL
LIN {X 0,Y 601.427,Z 307.07,A -85,B 0,C 180,E1 -699.478,E2 -699.478} C_VEL
LIN {X 0,Y 601.392,Z 307.067,A -85,B 0,C 180,E1 -702.312,E2 -702.312} C_VEL
LIN {X 0,Y 601.409,Z 307.065,A -85,B 0,C 180,E1 -704.409,E2 -704.409} C_VEL
LIN {X 0,Y 601.415,Z 307.074,A -85,B 0,C 180,E1 -707.172,E2 -707.172} C_VEL
LIN {X 0,Y 601.434,Z 307.062,A -85,B 0,C 180,E1 -709.905,E2 -709.905} C_VEL
LIN {X 0,Y 601.441,Z 307.065,A -85,B 0,C 180,E1 -712.615,E2 -712.615} C_VEL
LIN {X 0,Y 601.411,Z 307.069,A -85,B 0,C 180,E1 -715.308,E2 -715.308} C_VEL
LIN {X 0,Y 601.437,Z 307.062,A -85,B 0,C 180,E1 -717.991,E2 -717.991} C_VEL
LIN {X 0,Y 601.455,Z 307.067,A -85,B 0,C 180,E1 -720.67,E2 -720.67} C_VEL
LIN {X 0,Y 601.417,Z 307.066,A -85,B 0,C 180,E1 -723.35,E2 -723.35} C_VEL
LIN {X 0,Y 601.442,Z 307.062,A -85,B 0,C 180,E1 -726.037,E2 -726.037} C_VEL
LIN {X 0,Y 601.437,Z 307.07,A -85,B 0,C 180,E1 -728.738,E2 -728.738} C_VEL
LIN {X 0,Y 601.411,Z 307.065,A -85,B 0,C 180,E1 -731.459,E2 -731.459} C_VEL
LIN {X 0,Y 601.42,Z 307.069,A -85,B 0,C 180,E1 -734.206,E2 -734.206} C_VEL
LIN {X 0,Y 601.419,Z 307.066,A -85,B 0,C 180,E1 -736.987,E2 -736.987} C_VEL
LIN {X 0,Y 601.404,Z 307.068,A -85,B 0,C 180,E1 -739.81,E2 -739.81} C_VEL
LIN {X 0,Y 601.411,Z 307.068,A -85,B 0,C 180,E1 -742.683,E2 -742.683} C_VEL
LIN {X 0,Y 601.398,Z 307.068,A -85,B 0,C 180,E1 -744.879,E2 -744.879} C_VEL
LIN {X 0,Y 601.413,Z 307.065,A -85,B 0,C 180,E1 -747.362,E2 -747.362} C_VEL
LIN {X 0,Y 601.429,Z 307.072,A -85,B 0,C 180,E1 -750.164,E2 -750.164} C_VEL
LIN {X 0,Y 601.413,Z 307.066,A -85,B 0,C 180,E1 -752.714,E2 -752.714} C_VEL
LIN {X 0,Y 601.389,Z 307.068,A -85,B 0,C 180,E1 -755.111,E2 -755.111} C_VEL
LIN {X 0,Y 601.436,Z 307.065,A -85,B 0,C 180,E1 -757.419,E2 -757.419} C_VEL
LIN {X 0,Y 601.413,Z 307.073,A -85,B 0,C 180,E1 -759.995,E2 -759.995} C_VEL
LIN {X 0,Y 601.407,Z 307.066,A -85,B 0,C 180,E1 -762.671,E2 -762.671} C_VEL
LIN {X 0,Y 601.428,Z 307.07,A -85,B 0,C 180,E1 -765.482,E2 -765.482} C_VEL
LIN {X 0,Y 601.429,Z 307.067,A -85,B 0,C 180,E1 -766.428,E2 -766.428} C_VEL
LIN {X 0,Y 601.493,Z 307.667,A -85,B 0,C 180,E1 -767.401,E2 -767.401} C_VEL
LIN {X 0,Y 601.464,Z 312.149,A -85,B 0,C 180,E1 -770.009,E2 -770.009} C_VEL
LIN {X 0,Y 601.509,Z 316.937,A -85,B 0,C 180,E1 -772.609,E2 -772.609} C_VEL
LIN {X 0,Y 601.471,Z 321.813,A -85,B 0,C 180,E1 -775.072,E2 -775.072} C_VEL
LIN {X 0,Y 601.434,Z 326.847,A -85,B 0,C 180,E1 -777.485,E2 -777.485} C_VEL
LIN {X 0,Y 601.43,Z 332.026,A -85,B 0,C 180,E1 -779.852,E2 -779.852} C_VEL
LIN {X 0,Y 601.383,Z 337.326,A -85,B 0,C 180,E1 -782.131,E2 -782.131} C_VEL
LIN {X 0,Y 601.411,Z 342.716,A -85,B 0,C 180,E1 -784.382,E2 -784.382} C_VEL
LIN {X 0,Y 601.372,Z 349.902,A -85,B 0,C 180,E1 -787.316,E2 -787.316} C_VEL
LIN {X 0,Y 601.369,Z 357.088,A -85,B 0,C 180,E1 -790.189,E2 -790.189} C_VEL
LIN {X 0,Y 601.336,Z 364.274,A -85,B 0,C 180,E1 -793.011,E2 -793.011} C_VEL
LIN {X 0,Y 601.335,Z 371.46,A -85,B 0,C 180,E1 -795.793,E2 -795.793} C_VEL
LIN {X 0,Y 601.37,Z 377.579,A -85,B 0,C 180,E1 -798.113,E2 -798.113} C_VEL
LIN {X 0,Y 601.609,Z 387.254,A -85,B 0,C 180,E1 -798.31,E2 -798.31} C_VEL
LIN {X 0,Y 601.531,Z 399.26,A -85,B 0,C 180,E1 -798.656,E2 -798.656} C_VEL
LIN {X 0,Y 601.486,Z 411.437,A -85,B 0,C 180,E1 -799.141,E2 -799.141} C_VEL
LIN {X 0,Y 601.476,Z 422.757,A -85,B 0,C 180,E1 -799.736,E2 -799.736} C_VEL
LIN {X 0,Y 601.462,Z 434.248,A -85,B 0,C 180,E1 -800.5,E2 -800.5} C_VEL
LIN {X 0,Y 601.436,Z 443.521,A -85,B 0,C 180,E1 -801.262,E2 -801.262} C_VEL
LIN {X 0,Y 601.4,Z 451.994,A -85,B 0,C 180,E1 -802.108,E2 -802.108} C_VEL
LIN {X 0,Y 601.382,Z 460.239,A -85,B 0,C 180,E1 -803.12,E2 -803.12} C_VEL
LIN {X 0,Y 601.361,Z 465.868,A -85,B 0,C 180,E1 -803.962,E2 -803.962} C_VEL
LIN {X 0,Y 601.345,Z 471.365,A -85,B 0,C 180,E1 -804.971,E2 -804.971} C_VEL
LIN {X 0,Y 601.347,Z 475.672,A -85,B 0,C 180,E1 -805.979,E2 -805.979} C_VEL
LIN {X 0,Y 601.344,Z 477.959,A -85,B 0,C 180,E1 -806.65,E2 -806.65} C_VEL
LIN {X 0,Y 601.325,Z 479.805,A -85,B 0,C 180,E1 -807.32,E2 -807.32} C_VEL
LIN {X 0,Y 601.343,Z 481.199,A -85,B 0,C 180,E1 -807.991,E2 -807.991} C_VEL
LIN {X 0,Y 601.339,Z 482.783,A -85,B 0,C 180,E1 -809.33,E2 -809.33} C_VEL
LIN {X 0,Y 601.335,Z 482.991,A -85,B 0,C 180,E1 -810,E2 -810} C_VEL
LIN {X 0,Y 601.347,Z 482.185,A -85,B 0,C 180,E1 -811.339,E2 -811.339} C_VEL
LIN {X 0,Y 601.343,Z 481.199,A -85,B 0,C 180,E1 -812.009,E2 -812.009} C_VEL
LIN {X 0,Y 601.325,Z 479.805,A -85,B 0,C 180,E1 -812.68,E2 -812.68} C_VEL
LIN {X 0,Y 601.368,Z 476.894,A -85,B 0,C 180,E1 -813.685,E2 -813.685} C_VEL
LIN {X 0,Y 601.336,Z 472.949,A -85,B 0,C 180,E1 -814.693,E2 -814.693} C_VEL
LIN {X 0,Y 601.374,Z 467.857,A -85,B 0,C 180,E1 -815.701,E2 -815.701} C_VEL
LIN {X 0,Y 601.382,Z 461.47,A -85,B 0,C 180,E1 -816.711,E2 -816.711} C_VEL
LIN {X 0,Y 601.396,Z 453.482,A -85,B 0,C 180,E1 -817.723,E2 -817.723} C_VEL
LIN {X 0,Y 601.423,Z 445.341,A -85,B 0,C 180,E1 -818.568,E2 -818.568} C_VEL
LIN {X 0,Y 601.455,Z 435.386,A -85,B 0,C 180,E1 -819.415,E2 -819.415} C_VEL
LIN {X 0,Y 601.465,Z 425.572,A -85,B 0,C 180,E1 -820.094,E2 -820.094} C_VEL
LIN {X 0,Y 601.474,Z 414.928,A -85,B 0,C 180,E1 -820.69,E2 -820.69} C_VEL
LIN {X 0,Y 601.515,Z 401.857,A -85,B 0,C 180,E1 -821.253,E2 -821.253} C_VEL
LIN {X 0,Y 601.578,Z 389.045,A -85,B 0,C 180,E1 -821.647,E2 -821.647} C_VEL
LIN {X 0,Y 601.456,Z 378.412,A -85,B 0,C 180,E1 -821.872,E2 -821.872} C_VEL
LIN {X 0,Y 601.341,Z 377.467,A -85,B 0,C 180,E1 -821.909,E2 -821.909} C_VEL
LIN {X 0,Y 601.327,Z 369.664,A -85,B 0,C 180,E1 -824.899,E2 -824.899} C_VEL
LIN {X 0,Y 601.368,Z 362.478,A -85,B 0,C 180,E1 -827.689,E2 -827.689} C_VEL
LIN {X 0,Y 601.356,Z 355.291,A -85,B 0,C 180,E1 -830.524,E2 -830.524} C_VEL
LIN {X 0,Y 601.386,Z 348.105,A -85,B 0,C 180,E1 -833.412,E2 -833.412} C_VEL
LIN {X 0,Y 601.396,Z 342.125,A -85,B 0,C 180,E1 -835.863,E2 -835.863} C_VEL
LIN {X 0,Y 601.433,Z 335.151,A -85,B 0,C 180,E1 -838.788,E2 -838.788} C_VEL
LIN {X 0,Y 601.443,Z 329.137,A -85,B 0,C 180,E1 -841.458,E2 -841.458} C_VEL
LIN {X 0,Y 601.456,Z 323.483,A -85,B 0,C 180,E1 -844.116,E2 -844.116} C_VEL
LIN {X 0,Y 601.494,Z 318.523,A -85,B 0,C 180,E1 -846.576,E2 -846.576} C_VEL
LIN {X 0,Y 601.512,Z 313.712,A -85,B 0,C 180,E1 -849.119,E2 -849.119} C_VEL
LIN {X 0,Y 601.511,Z 309.077,A -85,B 0,C 180,E1 -851.757,E2 -851.757} C_VEL
LIN {X 0,Y 601.465,Z 307.554,A -85,B 0,C 180,E1 -852.665,E2 -852.665} C_VEL
LIN {X 0,Y 601.429,Z 307.069,A -85,B 0,C 180,E1 -853.586,E2 -853.586} C_VEL
LIN {X 0,Y 601.431,Z 307.07,A -85,B 0,C 180,E1 -856.427,E2 -856.427} C_VEL
LIN {X 0,Y 601.414,Z 307.065,A -85,B 0,C 180,E1 -859.125,E2 -859.125} C_VEL
LIN {X 0,Y 601.413,Z 307.069,A -85,B 0,C 180,E1 -861.731,E2 -861.731} C_VEL
LIN {X 0,Y 601.387,Z 307.075,A -85,B 0,C 180,E1 -864.245,E2 -864.245} C_VEL
LIN {X 0,Y 601.426,Z 307.064,A -85,B 0,C 180,E1 -866.686,E2 -866.686} C_VEL
LIN {X 0,Y 601.412,Z 307.065,A -85,B 0,C 180,E1 -869.057,E2 -869.057} C_VEL
LIN {X 0,Y 601.421,Z 307.066,A -85,B 0,C 180,E1 -871.372,E2 -871.372} C_VEL
LIN {X 0,Y 601.397,Z 307.074,A -85,B 0,C 180,E1 -873.636,E2 -873.636} C_VEL
LIN {X 0,Y 601.459,Z 307.068,A -85,B 0,C 180,E1 -875.859,E2 -875.859} C_VEL
LIN {X 0,Y 601.406,Z 307.065,A -85,B 0,C 180,E1 -878.76,E2 -878.76} C_VEL
LIN {X 0,Y 601.419,Z 307.074,A -85,B 0,C 180,E1 -881.608,E2 -881.608} C_VEL
LIN {X 0,Y 601.441,Z 307.069,A -85,B 0,C 180,E1 -883.713,E2 -883.713} C_VEL
LIN {X 0,Y 601.41,Z 307.065,A -85,B 0,C 180,E1 -886.484,E2 -886.484} C_VEL
LIN {X 0,Y 601.416,Z 307.071,A -85,B 0,C 180,E1 -889.224,E2 -889.224} C_VEL
LIN {X 0,Y 601.442,Z 307.063,A -85,B 0,C 180,E1 -891.939,E2 -891.939} C_VEL
LIN {X 0,Y 601.419,Z 307.065,A -85,B 0,C 180,E1 -894.635,E2 -894.635} C_VEL
LIN {X 0,Y 601.443,Z 307.07,A -85,B 0,C 180,E1 -897.321,E2 -897.321} C_VEL
LIN {X 0,Y 601.445,Z 307.061,A -85,B 0,C 180,E1 -900,E2 -900} C_VEL
LIN {X 0,Y 601.431,Z 307.066,A -85,B 0,C 180,E1 -902.679,E2 -902.679} C_VEL
LIN {X 0,Y 601.433,Z 307.067,A -85,B 0,C 180,E1 -905.364,E2 -905.364} C_VEL
LIN {X 0,Y 601.437,Z 307.061,A -85,B 0,C 180,E1 -908.06,E2 -908.06} C_VEL
LIN {X 0,Y 601.423,Z 307.072,A -85,B 0,C 180,E1 -911.012,E2 -911.012} C_VEL
LIN {X 0,Y 601.405,Z 307.068,A -85,B 0,C 180,E1 -912.364,E2 -912.364} C_VEL
LIN {X 0,Y 600.738,Z 307.158,A -85,B 0,C 180,E1 -912.923,E2 -912.923} C_VEL
LIN {X 0,Y 597.89,Z 307.515,A -85,B 0,C 180,E1 -913.831,E2 -913.831} C_VEL
LIN {X 0,Y 595.481,Z 307.813,A -85,B 0,C 180,E1 -914.561,E2 -914.561} C_VEL
LIN {X 0,Y 594.443,Z 307.938,A -85,B 0,C 180,E1 -915.125,E2 -915.125} C_VEL
LIN {X 0,Y 594.357,Z 307.946,A -85,B 0,C 180,E1 -915.316,E2 -915.316} C_VEL
LIN {X 0,Y 594.35,Z 307.945,A -85,B 0,C 180,E1 -917.905,E2 -917.905} C_VEL
LIN {X 0,Y 594.403,Z 307.946,A -85,B 0,C 180,E1 -920.775,E2 -920.775} C_VEL
LIN {X 0,Y 594.383,Z 307.94,A -85,B 0,C 180,E1 -923.704,E2 -923.704} C_VEL
LIN {X 0,Y 594.383,Z 307.948,A -85,B 0,C 180,E1 -926.699,E2 -926.699} C_VEL
LIN {X 0,Y 594.379,Z 307.943,A -85,B 0,C 180,E1 -928.998,E2 -928.998} C_VEL
LIN {X 0,Y 594.39,Z 307.94,A -85,B 0,C 180,E1 -931.645,E2 -931.645} C_VEL
LIN {X 0,Y 594.378,Z 307.947,A -85,B 0,C 180,E1 -934.58,E2 -934.58} C_VEL
LIN {X 0,Y 594.383,Z 307.941,A -85,B 0,C 180,E1 -937.086,E2 -937.086} C_VEL
LIN {X 0,Y 594.372,Z 307.945,A -85,B 0,C 180,E1 -939.774,E2 -939.774} C_VEL
LIN {X 0,Y 594.367,Z 307.949,A -85,B 0,C 180,E1 -942.375,E2 -942.375} C_VEL
LIN {X 0,Y 594.36,Z 307.943,A -85,B 0,C 180,E1 -945.191,E2 -945.191} C_VEL
LIN {X 0,Y 594.366,Z 307.946,A -85,B 0,C 180,E1 -947.625,E2 -947.625} C_VEL
LIN {X 0,Y 594.389,Z 307.944,A -85,B 0,C 180,E1 -950.321,E2 -950.321} C_VEL
LIN {X 0,Y 594.384,Z 307.94,A -85,B 0,C 180,E1 -952.913,E2 -952.913} C_VEL
LIN {X 0,Y 594.378,Z 307.951,A -85,B 0,C 180,E1 -955.861,E2 -955.861} C_VEL
LIN {X 0,Y 594.387,Z 307.94,A -85,B 0,C 180,E1 -958.651,E2 -958.651} C_VEL
LIN {X 0,Y 594.38,Z 307.942,A -85,B 0,C 180,E1 -961.042,E2 -961.042} C_VEL
LIN {X 0,Y 594.386,Z 307.944,A -85,B 0,C 180,E1 -963.976,E2 -963.976} C_VEL
LIN {X 0,Y 594.386,Z 307.941,A -85,B 0,C 180,E1 -966.296,E2 -966.296} C_VEL
LIN {X 0,Y 594.404,Z 307.943,A -85,B 0,C 180,E1 -969.225,E2 -969.225} C_VEL
LIN {X 0,Y 594.352,Z 307.946,A -85,B 0,C 180,E1 -972.095,E2 -972.095} C_VEL
LIN {X 0,Y 594.364,Z 307.943,A -85,B 0,C 180,E1 -974.219,E2 -974.219} C_VEL
LIN {X 0,Y 594.365,Z 307.948,A -85,B 0,C 180,E1 -977.017,E2 -977.017} C_VEL
LIN {X 0,Y 594.396,Z 307.941,A -85,B 0,C 180,E1 -979.784,E2 -979.784} C_VEL
LIN {X 0,Y 594.389,Z 307.941,A -85,B 0,C 180,E1 -982.527,E2 -982.527} C_VEL
LIN {X 0,Y 594.388,Z 307.948,A -85,B 0,C 180,E1 -985.252,E2 -985.252} C_VEL
LIN {X 0,Y 594.406,Z 307.938,A -85,B 0,C 180,E1 -987.967,E2 -987.967} C_VEL
LIN {X 0,Y 594.418,Z 307.942,A -85,B 0,C 180,E1 -990.677,E2 -990.677} C_VEL
LIN {X 0,Y 594.377,Z 307.944,A -85,B 0,C 180,E1 -993.389,E2 -993.389} C_VEL
LIN {X 0,Y 594.392,Z 307.94,A -85,B 0,C 180,E1 -996.109,E2 -996.109} C_VEL
LIN {X 0,Y 594.394,Z 307.949,A -85,B 0,C 180,E1 -998.842,E2 -998.842} C_VEL
LIN {X 0,Y 594.391,Z 307.94,A -85,B 0,C 180,E1 -1001.596,E2 -1001.596} C_VEL
LIN {X 0,Y 594.387,Z 307.946,A -85,B 0,C 180,E1 -1004.377,E2 -1004.377} C_VEL
LIN {X 0,Y 594.387,Z 307.942,A -85,B 0,C 180,E1 -1007.193,E2 -1007.193} C_VEL
LIN {X 0,Y 594.374,Z 307.944,A -85,B 0,C 180,E1 -1010.054,E2 -1010.054} C_VEL
LIN {X 0,Y 594.361,Z 307.945,A -85,B 0,C 180,E1 -1012.967,E2 -1012.967} C_VEL
LIN {X 0,Y 594.373,Z 307.942,A -85,B 0,C 180,E1 -1015.193,E2 -1015.193} C_VEL
LIN {X 0,Y 594.382,Z 307.941,A -85,B 0,C 180,E1 -1017.527,E2 -1017.527} C_VEL
LIN {X 0,Y 594.384,Z 307.949,A -85,B 0,C 180,E1 -1020.329,E2 -1020.329} C_VEL
LIN {X 0,Y 594.376,Z 307.942,A -85,B 0,C 180,E1 -1022.95,E2 -1022.95} C_VEL
LIN {X 0,Y 594.351,Z 307.945,A -85,B 0,C 180,E1 -1025.409,E2 -1025.409} C_VEL
LIN {X 0,Y 594.386,Z 307.948,A -85,B 0,C 180,E1 -1027.94,E2 -1027.94} C_VEL
LIN {X 0,Y 594.378,Z 307.941,A -85,B 0,C 180,E1 -1030.823,E2 -1030.823} C_VEL
LIN {X 0,Y 594.38,Z 307.949,A -85,B 0,C 180,E1 -1033.841,E2 -1033.841} C_VEL
LIN {X 0,Y 594.377,Z 307.941,A -85,B 0,C 180,E1 -1036.702,E2 -1036.702} C_VEL
LIN {X 0,Y 594.371,Z 307.946,A -85,B 0,C 180,E1 -1039.434,E2 -1039.434} C_VEL
LIN {X 0,Y 594.388,Z 307.941,A -85,B 0,C 180,E1 -1042.391,E2 -1042.391} C_VEL
LIN {X 0,Y 594.378,Z 307.947,A -85,B 0,C 180,E1 -1045.42,E2 -1045.42} C_VEL
LIN {X 0,Y 594.389,Z 307.94,A -85,B 0,C 180,E1 -1048.355,E2 -1048.355} C_VEL
LIN {X 0,Y 594.382,Z 307.943,A -85,B 0,C 180,E1 -1051.042,E2 -1051.042} C_VEL
LIN {X 0,Y 594.382,Z 307.943,A -85,B 0,C 180,E1 -1053.978,E2 -1053.978} C_VEL
LIN {X 0,Y 594.384,Z 307.94,A -85,B 0,C 180,E1 -1056.296,E2 -1056.296} C_VEL
LIN {X 0,Y 594.403,Z 307.946,A -85,B 0,C 180,E1 -1059.225,E2 -1059.225} C_VEL
LIN {X 0,Y 594.35,Z 307.945,A -85,B 0,C 180,E1 -1062.095,E2 -1062.095} C_VEL
LIN {X 0,Y 594.362,Z 307.943,A -85,B 0,C 180,E1 -1064.219,E2 -1064.219} C_VEL
LIN {X 0,Y 594.381,Z 307.941,A -85,B 0,C 180,E1 -1066.321,E2 -1066.321} C_VEL
LIN {X 0,Y 594.373,Z 307.952,A -85,B 0,C 180,E1 -1069.095,E2 -1069.095} C_VEL
LIN {X 0,Y 594.41,Z 307.937,A -85,B 0,C 180,E1 -1071.844,E2 -1071.844} C_VEL
LIN {X 0,Y 594.399,Z 307.942,A -85,B 0,C 180,E1 -1074.573,E2 -1074.573} C_VEL
LIN {X 0,Y 594.398,Z 307.942,A -85,B 0,C 180,E1 -1077.29,E2 -1077.29} C_VEL
LIN {X 0,Y 594.414,Z 307.937,A -85,B 0,C 180,E1 -1080,E2 -1080} C_VEL
LIN {X 0,Y 594.408,Z 307.947,A -85,B 0,C 180,E1 -1082.711,E2 -1082.711} C_VEL
LIN {X 0,Y 594.388,Z 307.94,A -85,B 0,C 180,E1 -1085.428,E2 -1085.428} C_VEL
LIN {X 0,Y 594.418,Z 307.939,A -85,B 0,C 180,E1 -1088.157,E2 -1088.157} C_VEL
LIN {X 0,Y 594.389,Z 307.942,A -85,B 0,C 180,E1 -1091.074,E2 -1091.074} C_VEL
LIN {X 0,Y 594.378,Z 307.941,A -85,B 0,C 180,E1 -1093.679,E2 -1093.679} C_VEL
LIN {X 0,Y 594.392,Z 307.944,A -85,B 0,C 180,E1 -1096.719,E2 -1096.719} C_VEL
LIN {X 0,Y 594.366,Z 307.942,A -85,B 0,C 180,E1 -1099.335,E2 -1099.335} C_VEL
LIN {X 0,Y 594.367,Z 307.943,A -85,B 0,C 180,E1 -1101.504,E2 -1101.504} C_VEL
LIN {X 0,Y 594.389,Z 307.946,A -85,B 0,C 180,E1 -1104.446,E2 -1104.446} C_VEL
LIN {X 0,Y 594.379,Z 307.943,A -85,B 0,C 180,E1 -1106.7,E2 -1106.7} C_VEL
LIN {X 0,Y 594.38,Z 307.941,A -85,B 0,C 180,E1 -1108.999,E2 -1108.999} C_VEL
LIN {X 0,Y 594.376,Z 307.945,A -85,B 0,C 180,E1 -1111.643,E2 -1111.643} C_VEL
LIN {X 0,Y 594.375,Z 307.943,A -85,B 0,C 180,E1 -1114.581,E2 -1114.581} C_VEL
LIN {X 0,Y 594.39,Z 307.945,A -85,B 0,C 180,E1 -1117.609,E2 -1117.609} C_VEL
LIN {X 0,Y 594.364,Z 307.944,A -85,B 0,C 180,E1 -1120.568,E2 -1120.568} C_VEL
LIN {X 0,Y 594.367,Z 307.946,A -85,B 0,C 180,E1 -1123.3,E2 -1123.3} C_VEL
LIN {X 0,Y 594.369,Z 307.951,A -85,B 0,C 180,E1 -1126.161,E2 -1126.161} C_VEL
LIN {X 0,Y 594.38,Z 307.946,A -85,B 0,C 180,E1 -1126.702,E2 -1126.702} C_VEL
LIN {X 0,Y 594.516,Z 310.864,A -85,B 0,C 180,E1 -1128.548,E2 -1128.548} C_VEL
LIN {X 0,Y 594.512,Z 315.646,A -85,B 0,C 180,E1 -1131.281,E2 -1131.281} C_VEL
LIN {X 0,Y 594.472,Z 320.352,A -85,B 0,C 180,E1 -1133.764,E2 -1133.764} C_VEL
LIN {X 0,Y 594.444,Z 325.296,A -85,B 0,C 180,E1 -1136.243,E2 -1136.243} C_VEL
LIN {X 0,Y 594.403,Z 330.369,A -85,B 0,C 180,E1 -1138.652,E2 -1138.652} C_VEL
LIN {X 0,Y 594.383,Z 335.678,A -85,B 0,C 180,E1 -1141.043,E2 -1141.043} C_VEL
LIN {X 0,Y 594.336,Z 342.716,A -85,B 0,C 180,E1 -1144.054,E2 -1144.054} C_VEL
LIN {X 0,Y 594.307,Z 348.105,A -85,B 0,C 180,E1 -1146.293,E2 -1146.293} C_VEL
LIN {X 0,Y 594.303,Z 355.001,A -85,B 0,C 180,E1 -1149.104,E2 -1149.104} C_VEL
LIN {X 0,Y 594.277,Z 360.681,A -85,B 0,C 180,E1 -1151.379,E2 -1151.379} C_VEL
LIN {X 0,Y 594.262,Z 367.867,A -85,B 0,C 180,E1 -1154.216,E2 -1154.216} C_VEL
LIN {X 0,Y 594.22,Z 375.053,A -85,B 0,C 180,E1 -1157.014,E2 -1157.014} C_VEL
LIN {X 0,Y 594.269,Z 377.528,A -85,B 0,C 180,E1 -1157.969,E2 -1157.969} C_VEL
LIN {X 0,Y 594.653,Z 382.396,A -85,B 0,C 180,E1 -1158.064,E2 -1158.064} C_VEL
LIN {X 0,Y 594.582,Z 395.84,A -85,B 0,C 180,E1 -1158.408,E2 -1158.408} C_VEL
LIN {X 0,Y 594.521,Z 408.058,A -85,B 0,C 180,E1 -1158.864,E2 -1158.864} C_VEL
LIN {X 0,Y 594.475,Z 419.771,A -85,B 0,C 180,E1 -1159.441,E2 -1159.441} C_VEL
LIN {X 0,Y 594.453,Z 430.748,A -85,B 0,C 180,E1 -1160.129,E2 -1160.129} C_VEL
LIN {X 0,Y 594.404,Z 441.586,A -85,B 0,C 180,E1 -1160.987,E2 -1160.987} C_VEL
LIN {X 0,Y 594.365,Z 450.396,A -85,B 0,C 180,E1 -1161.843,E2 -1161.843} C_VEL
LIN {X 0,Y 594.305,Z 459.004,A -85,B 0,C 180,E1 -1162.867,E2 -1162.867} C_VEL
LIN {X 0,Y 594.289,Z 465.87,A -85,B 0,C 180,E1 -1163.89,E2 -1163.89} C_VEL
LIN {X 0,Y 594.254,Z 471.364,A -85,B 0,C 180,E1 -1164.911,E2 -1164.911} C_VEL
LIN {X 0,Y 594.262,Z 475.669,A -85,B 0,C 180,E1 -1165.931,E2 -1165.931} C_VEL
LIN {X 0,Y 594.267,Z 477.961,A -85,B 0,C 180,E1 -1166.61,E2 -1166.61} C_VEL
LIN {X 0,Y 594.225,Z 479.8,A -85,B 0,C 180,E1 -1167.288,E2 -1167.288} C_VEL
LIN {X 0,Y 594.242,Z 481.194,A -85,B 0,C 180,E1 -1167.967,E2 -1167.967} C_VEL
LIN {X 0,Y 594.247,Z 482.187,A -85,B 0,C 180,E1 -1168.645,E2 -1168.645} C_VEL
LIN {X 0,Y 594.239,Z 482.783,A -85,B 0,C 180,E1 -1169.322,E2 -1169.322} C_VEL
LIN {X 0,Y 594.236,Z 482.984,A -85,B 0,C 180,E1 -1170,E2 -1170} C_VEL
LIN {X 0,Y 594.239,Z 482.783,A -85,B 0,C 180,E1 -1170.678,E2 -1170.678} C_VEL
LIN {X 0,Y 594.247,Z 482.187,A -85,B 0,C 180,E1 -1171.355,E2 -1171.355} C_VEL
LIN {X 0,Y 594.242,Z 481.194,A -85,B 0,C 180,E1 -1172.033,E2 -1172.033} C_VEL
LIN {X 0,Y 594.225,Z 479.8,A -85,B 0,C 180,E1 -1172.712,E2 -1172.712} C_VEL
LIN {X 0,Y 594.289,Z 476.89,A -85,B 0,C 180,E1 -1173.729,E2 -1173.729} C_VEL
LIN {X 0,Y 594.241,Z 472.943,A -85,B 0,C 180,E1 -1174.749,E2 -1174.749} C_VEL
LIN {X 0,Y 594.3,Z 467.849,A -85,B 0,C 180,E1 -1175.769,E2 -1175.769} C_VEL
LIN {X 0,Y 594.316,Z 461.465,A -85,B 0,C 180,E1 -1176.791,E2 -1176.791} C_VEL
LIN {X 0,Y 594.346,Z 453.485,A -85,B 0,C 180,E1 -1177.816,E2 -1177.816} C_VEL
LIN {X 0,Y 594.378,Z 445.344,A -85,B 0,C 180,E1 -1178.671,E2 -1178.671} C_VEL
LIN {X 0,Y 594.418,Z 435.374,A -85,B 0,C 180,E1 -1179.528,E2 -1179.528} C_VEL
LIN {X 0,Y 594.455,Z 425.558,A -85,B 0,C 180,E1 -1180.215,E2 -1180.215} C_VEL
LIN {X 0,Y 594.494,Z 414.933,A -85,B 0,C 180,E1 -1180.817,E2 -1180.817} C_VEL
LIN {X 0,Y 594.545,Z 402.199,A -85,B 0,C 180,E1 -1181.374,E2 -1181.374} C_VEL
LIN {X 0,Y 594.632,Z 389.889,A -85,B 0,C 180,E1 -1181.764,E2 -1181.764} C_VEL
LIN {X 0,Y 594.531,Z 379.286,A -85,B 0,C 180,E1 -1181.997,E2 -1181.997} C_VEL
LIN {X 0,Y 594.273,Z 377.467,A -85,B 0,C 180,E1 -1182.052,E2 -1182.052} C_VEL
LIN {X 0,Y 594.253,Z 369.664,A -85,B 0,C 180,E1 -1185.081,E2 -1185.081} C_VEL
LIN {X 0,Y 594.275,Z 362.478,A -85,B 0,C 180,E1 -1187.907,E2 -1187.907} C_VEL
LIN {X 0,Y 594.302,Z 355.291,A -85,B 0,C 180,E1 -1190.779,E2 -1190.779} C_VEL
LIN {X 0,Y 594.303,Z 349.902,A -85,B 0,C 180,E1 -1192.97,E2 -1192.97} C_VEL
LIN {X 0,Y 594.334,Z 344.512,A -85,B 0,C 180,E1 -1195.195,E2 -1195.195} C_VEL
LIN {X 0,Y 594.344,Z 338.991,A -85,B 0,C 180,E1 -1197.518,E2 -1197.518} C_VEL
LIN {X 0,Y 594.389,Z 332.576,A -85,B 0,C 180,E1 -1200.328,E2 -1200.328} C_VEL
LIN {X 0,Y 594.423,Z 326.974,A -85,B 0,C 180,E1 -1202.947,E2 -1202.947} C_VEL
LIN {X 0,Y 594.455,Z 321.965,A -85,B 0,C 180,E1 -1205.402,E2 -1205.402} C_VEL
LIN {X 0,Y 594.495,Z 317.086,A -85,B 0,C 180,E1 -1207.932,E2 -1207.932} C_VEL
LIN {X 0,Y 594.52,Z 311.918,A -85,B 0,C 180,E1 -1210.837,E2 -1210.837} C_VEL
LIN {X 0,Y 594.44,Z 308.539,A -85,B 0,C 180,E1 -1212.86,E2 -1212.86} C_VEL
LIN {X 0,Y 594.38,Z 307.949,A -85,B 0,C 180,E1 -1213.298,E2 -1213.298} C_VEL
LIN {X 0,Y 594.362,Z 307.953,A -85,B 0,C 180,E1 -1216.161,E2 -1216.161} C_VEL
LIN {X 0,Y 594.381,Z 307.946,A -85,B 0,C 180,E1 -1218.536,E2 -1218.536} C_VEL
LIN {X 0,Y 594.379,Z 307.942,A -85,B 0,C 180,E1 -1221.296,E2 -1221.296} C_VEL
LIN {X 0,Y 594.351,Z 307.95,A -85,B 0,C 180,E1 -1223.755,E2 -1223.755} C_VEL
LIN {X 0,Y 594.379,Z 307.947,A -85,B 0,C 180,E1 -1226.238,E2 -1226.238} C_VEL
LIN {X 0,Y 594.369,Z 307.943,A -85,B 0,C 180,E1 -1228.649,E2 -1228.649} C_VEL
LIN {X 0,Y 594.381,Z 307.941,A -85,B 0,C 180,E1 -1231.042,E2 -1231.042} C_VEL
LIN {X 0,Y 594.385,Z 307.947,A -85,B 0,C 180,E1 -1233.977,E2 -1233.977} C_VEL
LIN {X 0,Y 594.378,Z 307.943,A -85,B 0,C 180,E1 -1236.295,E2 -1236.295} C_VEL
LIN {X 0,Y 594.399,Z 307.941,A -85,B 0,C 180,E1 -1239.224,E2 -1239.224} C_VEL
LIN {X 0,Y 594.35,Z 307.947,A -85,B 0,C 180,E1 -1242.095,E2 -1242.095} C_VEL
LIN {X 0,Y 594.364,Z 307.944,A -85,B 0,C 180,E1 -1244.219,E2 -1244.219} C_VEL
LIN {X 0,Y 594.378,Z 307.941,A -85,B 0,C 180,E1 -1246.321,E2 -1246.321} C_VEL
LIN {X 0,Y 594.374,Z 307.946,A -85,B 0,C 180,E1 -1249.094,E2 -1249.094} C_VEL
LIN {X 0,Y 594.418,Z 307.939,A -85,B 0,C 180,E1 -1251.843,E2 -1251.843} C_VEL
LIN {X 0,Y 594.387,Z 307.94,A -85,B 0,C 180,E1 -1254.572,E2 -1254.572} C_VEL
LIN {X 0,Y 594.408,Z 307.947,A -85,B 0,C 180,E1 -1257.289,E2 -1257.289} C_VEL
LIN {X 0,Y 594.414,Z 307.937,A -85,B 0,C 180,E1 -1260,E2 -1260} C_VEL
LIN {X 0,Y 594.398,Z 307.942,A -85,B 0,C 180,E1 -1262.71,E2 -1262.71} C_VEL
LIN {X 0,Y 594.399,Z 307.942,A -85,B 0,C 180,E1 -1265.427,E2 -1265.427} C_VEL
LIN {X 0,Y 594.41,Z 307.937,A -85,B 0,C 180,E1 -1268.156,E2 -1268.156} C_VEL
LIN {X 0,Y 594.387,Z 307.947,A -85,B 0,C 180,E1 -1271.073,E2 -1271.073} C_VEL
LIN {X 0,Y 594.381,Z 307.941,A -85,B 0,C 180,E1 -1273.679,E2 -1273.679} C_VEL
LIN {X 0,Y 594.357,Z 307.946,A -85,B 0,C 180,E1 -1275.316,E2 -1275.316} C_VEL
LIN {X 0,Y 593.682,Z 308.03,A -85,B 0,C 180,E1 -1275.881,E2 -1275.881} C_VEL
LIN {X 0,Y 590.816,Z 308.395,A -85,B 0,C 180,E1 -1276.799,E2 -1276.799} C_VEL
LIN {X 0,Y 588.406,Z 308.69,A -85,B 0,C 180,E1 -1277.538,E2 -1277.538} C_VEL
LIN {X 0,Y 587.384,Z 308.814,A -85,B 0,C 180,E1 -1278.108,E2 -1278.108} C_VEL
LIN {X 0,Y 587.307,Z 308.824,A -85,B 0,C 180,E1 -1278.301,E2 -1278.301} C_VEL
LIN {X 0,Y 587.328,Z 308.823,A -85,B 0,C 180,E1 -1281.037,E2 -1281.037} C_VEL
LIN {X 0,Y 587.319,Z 308.822,A -85,B 0,C 180,E1 -1283.258,E2 -1283.258} C_VEL
LIN {X 0,Y 587.332,Z 308.819,A -85,B 0,C 180,E1 -1285.516,E2 -1285.516} C_VEL
LIN {X 0,Y 587.345,Z 308.818,A -85,B 0,C 180,E1 -1287.817,E2 -1287.817} C_VEL
LIN {X 0,Y 587.338,Z 308.827,A -85,B 0,C 180,E1 -1290.51,E2 -1290.51} C_VEL
LIN {X 0,Y 587.337,Z 308.819,A -85,B 0,C 180,E1 -1293.112,E2 -1293.112} C_VEL
LIN {X 0,Y 587.308,Z 308.825,A -85,B 0,C 180,E1 -1295.898,E2 -1295.898} C_VEL
LIN {X 0,Y 587.331,Z 308.825,A -85,B 0,C 180,E1 -1298.479,E2 -1298.479} C_VEL
LIN {X 0,Y 587.334,Z 308.818,A -85,B 0,C 180,E1 -1301.156,E2 -1301.156} C_VEL
LIN {X 0,Y 587.331,Z 308.829,A -85,B 0,C 180,E1 -1304.114,E2 -1304.114} C_VEL
LIN {X 0,Y 587.318,Z 308.82,A -85,B 0,C 180,E1 -1306.994,E2 -1306.994} C_VEL
LIN {X 0,Y 587.317,Z 308.827,A -85,B 0,C 180,E1 -1309.746,E2 -1309.746} C_VEL
LIN {X 0,Y 587.344,Z 308.82,A -85,B 0,C 180,E1 -1312.392,E2 -1312.392} C_VEL
LIN {X 0,Y 587.322,Z 308.82,A -85,B 0,C 180,E1 -1314.944,E2 -1314.944} C_VEL
LIN {X 0,Y 587.337,Z 308.822,A -85,B 0,C 180,E1 -1317.421,E2 -1317.421} C_VEL
LIN {X 0,Y 587.332,Z 308.827,A -85,B 0,C 180,E1 -1319.83,E2 -1319.83} C_VEL
LIN {X 0,Y 587.348,Z 308.818,A -85,B 0,C 180,E1 -1322.307,E2 -1322.307} C_VEL
LIN {X 0,Y 587.333,Z 308.819,A -85,B 0,C 180,E1 -1324.483,E2 -1324.483} C_VEL
LIN {X 0,Y 587.337,Z 308.827,A -85,B 0,C 180,E1 -1327.486,E2 -1327.486} C_VEL
LIN {X 0,Y 587.341,Z 308.818,A -85,B 0,C 180,E1 -1330.425,E2 -1330.425} C_VEL
LIN {X 0,Y 587.349,Z 308.826,A -85,B 0,C 180,E1 -1333.311,E2 -1333.311} C_VEL
LIN {X 0,Y 587.356,Z 308.816,A -85,B 0,C 180,E1 -1336.154,E2 -1336.154} C_VEL
LIN {X 0,Y 587.341,Z 308.823,A -85,B 0,C 180,E1 -1338.962,E2 -1338.962} C_VEL
LIN {X 0,Y 587.368,Z 308.817,A -85,B 0,C 180,E1 -1341.745,E2 -1341.745} C_VEL
LIN {X 0,Y 587.361,Z 308.817,A -85,B 0,C 180,E1 -1344.507,E2 -1344.507} C_VEL
LIN {X 0,Y 587.37,Z 308.821,A -85,B 0,C 180,E1 -1347.257,E2 -1347.257} C_VEL
LIN {X 0,Y 587.382,Z 308.813,A -85,B 0,C 180,E1 -1350,E2 -1350} C_VEL
LIN {X 0,Y 587.37,Z 308.821,A -85,B 0,C 180,E1 -1352.743,E2 -1352.743} C_VEL
LIN {X 0,Y 587.361,Z 308.817,A -85,B 0,C 180,E1 -1355.493,E2 -1355.493} C_VEL
LIN {X 0,Y 587.368,Z 308.817,A -85,B 0,C 180,E1 -1358.255,E2 -1358.255} C_VEL
LIN {X 0,Y 587.345,Z 308.821,A -85,B 0,C 180,E1 -1361.134,E2 -1361.134} C_VEL
LIN {X 0,Y 587.362,Z 308.819,A -85,B 0,C 180,E1 -1364.261,E2 -1364.261} C_VEL
LIN {X 0,Y 587.347,Z 308.817,A -85,B 0,C 180,E1 -1367.406,E2 -1367.406} C_VEL
LIN {X 0,Y 587.329,Z 308.826,A -85,B 0,C 180,E1 -1370.305,E2 -1370.305} C_VEL
LIN {X 0,Y 587.319,Z 308.821,A -85,B 0,C 180,E1 -1373.259,E2 -1373.259} C_VEL
LIN {X 0,Y 587.333,Z 308.819,A -85,B 0,C 180,E1 -1375.517,E2 -1375.517} C_VEL
LIN {X 0,Y 587.346,Z 308.819,A -85,B 0,C 180,E1 -1377.818,E2 -1377.818} C_VEL
LIN {X 0,Y 587.339,Z 308.824,A -85,B 0,C 180,E1 -1380.511,E2 -1380.511} C_VEL
LIN {X 0,Y 587.337,Z 308.818,A -85,B 0,C 180,E1 -1383.112,E2 -1383.112} C_VEL
LIN {X 0,Y 587.315,Z 308.827,A -85,B 0,C 180,E1 -1385.898,E2 -1385.898} C_VEL
LIN {X 0,Y 587.331,Z 308.822,A -85,B 0,C 180,E1 -1388.479,E2 -1388.479} C_VEL
LIN {X 0,Y 587.335,Z 308.818,A -85,B 0,C 180,E1 -1391.157,E2 -1391.157} C_VEL
LIN {X 0,Y 587.331,Z 308.826,A -85,B 0,C 180,E1 -1394.114,E2 -1394.114} C_VEL
LIN {X 0,Y 587.319,Z 308.82,A -85,B 0,C 180,E1 -1396.995,E2 -1396.995} C_VEL
LIN {X 0,Y 587.317,Z 308.83,A -85,B 0,C 180,E1 -1399.746,E2 -1399.746} C_VEL
LIN {X 0,Y 587.343,Z 308.818,A -85,B 0,C 180,E1 -1402.393,E2 -1402.393} C_VEL
LIN {X 0,Y 587.358,Z 308.823,A -85,B 0,C 180,E1 -1405.78,E2 -1405.78} C_VEL
LIN {X 0,Y 587.351,Z 308.818,A -85,B 0,C 180,E1 -1408.232,E2 -1408.232} C_VEL
LIN {X 0,Y 587.347,Z 308.818,A -85,B 0,C 180,E1 -1410.867,E2 -1410.867} C_VEL
LIN {X 0,Y 587.356,Z 308.82,A -85,B 0,C 180,E1 -1413.819,E2 -1413.819} C_VEL
LIN {X 0,Y 587.332,Z 308.82,A -85,B 0,C 180,E1 -1415.994,E2 -1415.994} C_VEL
LIN {X 0,Y 587.322,Z 308.82,A -85,B 0,C 180,E1 -1418.226,E2 -1418.226} C_VEL
LIN {X 0,Y 587.348,Z 308.825,A -85,B 0,C 180,E1 -1421.152,E2 -1421.152} C_VEL
LIN {X 0,Y 587.32,Z 308.82,A -85,B 0,C 180,E1 -1424.025,E2 -1424.025} C_VEL
LIN {X 0,Y 587.358,Z 308.815,A -85,B 0,C 180,E1 -1426.155,E2 -1426.155} C_VEL
LIN {X 0,Y 587.339,Z 308.826,A -85,B 0,C 180,E1 -1428.963,E2 -1428.963} C_VEL
LIN {X 0,Y 587.362,Z 308.816,A -85,B 0,C 180,E1 -1431.745,E2 -1431.745} C_VEL
LIN {X 0,Y 587.365,Z 308.818,A -85,B 0,C 180,E1 -1434.507,E2 -1434.507} C_VEL
LIN {X 0,Y 587.366,Z 308.819,A -85,B 0,C 180,E1 -1437.257,E2 -1437.257} C_VEL
LIN {X 0,Y 587.383,Z 308.813,A -85,B 0,C 180,E1 -1440,E2 -1440} C_VEL
LIN {X 0,Y 587.373,Z 308.824,A -85,B 0,C 180,E1 -1442.744,E2 -1442.744} C_VEL
LIN {X 0,Y 587.356,Z 308.816,A -85,B 0,C 180,E1 -1445.493,E2 -1445.493} C_VEL
LIN {X 0,Y 587.371,Z 308.818,A -85,B 0,C 180,E1 -1448.256,E2 -1448.256} C_VEL
LIN {X 0,Y 587.348,Z 308.818,A -85,B 0,C 180,E1 -1451.134,E2 -1451.134} C_VEL
LIN {X 0,Y 587.365,Z 308.821,A -85,B 0,C 180,E1 -1454.261,E2 -1454.261} C_VEL
LIN {X 0,Y 587.345,Z 308.817,A -85,B 0,C 180,E1 -1457.406,E2 -1457.406} C_VEL
LIN {X 0,Y 587.327,Z 308.829,A -85,B 0,C 180,E1 -1460.305,E2 -1460.305} C_VEL
LIN {X 0,Y 587.315,Z 308.821,A -85,B 0,C 180,E1 -1463.259,E2 -1463.259} C_VEL
LIN {X 0,Y 587.334,Z 308.819,A -85,B 0,C 180,E1 -1465.517,E2 -1465.517} C_VEL
LIN {X 0,Y 587.346,Z 308.822,A -85,B 0,C 180,E1 -1467.818,E2 -1467.818} C_VEL
LIN {X 0,Y 587.336,Z 308.822,A -85,B 0,C 180,E1 -1470.51,E2 -1470.51} C_VEL
LIN {X 0,Y 587.335,Z 308.82,A -85,B 0,C 180,E1 -1473.397,E2 -1473.397} C_VEL
LIN {X 0,Y 587.291,Z 308.833,A -85,B 0,C 180,E1 -1475.9,E2 -1475.9} C_VEL
LIN {X 0,Y 587.326,Z 308.822,A -85,B 0,C 180,E1 -1478.48,E2 -1478.48} C_VEL
LIN {X 0,Y 587.336,Z 308.82,A -85,B 0,C 180,E1 -1481.157,E2 -1481.157} C_VEL
LIN {X 0,Y 587.313,Z 308.828,A -85,B 0,C 180,E1 -1484.112,E2 -1484.112} C_VEL
LIN {X 0,Y 587.324,Z 308.829,A -85,B 0,C 180,E1 -1486.05,E2 -1486.05} C_VEL
LIN {X 0,Y 587.446,Z 309.575,A -85,B 0,C 180,E1 -1487.006,E2 -1487.006} C_VEL
LIN {X 0,Y 587.533,Z 312.687,A -85,B 0,C 180,E1 -1488.903,E2 -1488.903} C_VEL
LIN {X 0,Y 587.494,Z 317.296,A -85,B 0,C 180,E1 -1491.534,E2 -1491.534} C_VEL
LIN {X 0,Y 587.444,Z 322.14,A -85,B 0,C 180,E1 -1494.111,E2 -1494.111} C_VEL
LIN {X 0,Y 587.399,Z 327.665,A -85,B 0,C 180,E1 -1496.88,E2 -1496.88} C_VEL
LIN {X 0,Y 587.34,Z 333.889,A -85,B 0,C 180,E1 -1499.83,E2 -1499.83} C_VEL
LIN {X 0,Y 587.3,Z 339.495,A -85,B 0,C 180,E1 -1502.317,E2 -1502.317} C_VEL
LIN {X 0,Y 587.293,Z 346.309,A -85,B 0,C 180,E1 -1505.239,E2 -1505.239} C_VEL
LIN {X 0,Y 587.242,Z 353.495,A -85,B 0,C 180,E1 -1508.223,E2 -1508.223} C_VEL
LIN {X 0,Y 587.235,Z 360.681,A -85,B 0,C 180,E1 -1511.148,E2 -1511.148} C_VEL
LIN {X 0,Y 587.181,Z 367.867,A -85,B 0,C 180,E1 -1514.021,E2 -1514.021} C_VEL
LIN {X 0,Y 587.156,Z 375.053,A -85,B 0,C 180,E1 -1516.855,E2 -1516.855} C_VEL
LIN {X 0,Y 587.148,Z 377.523,A -85,B 0,C 180,E1 -1517.821,E2 -1517.821} C_VEL
LIN {X 0,Y 587.723,Z 382.403,A -85,B 0,C 180,E1 -1517.921,E2 -1517.921} C_VEL
LIN {X 0,Y 587.622,Z 395.825,A -85,B 0,C 180,E1 -1518.269,E2 -1518.269} C_VEL
LIN {X 0,Y 587.544,Z 407.709,A -85,B 0,C 180,E1 -1518.715,E2 -1518.715} C_VEL
LIN {X 0,Y 587.493,Z 419.77,A -85,B 0,C 180,E1 -1519.314,E2 -1519.314} C_VEL
LIN {X 0,Y 587.453,Z 430.748,A -85,B 0,C 180,E1 -1520.01,E2 -1520.01} C_VEL
LIN {X 0,Y 587.384,Z 439.641,A -85,B 0,C 180,E1 -1520.705,E2 -1520.705} C_VEL
LIN {X 0,Y 587.32,Z 448.764,A -85,B 0,C 180,E1 -1521.571,E2 -1521.571} C_VEL
LIN {X 0,Y 587.271,Z 456.313,A -85,B 0,C 180,E1 -1522.436,E2 -1522.436} C_VEL
LIN {X 0,Y 587.213,Z 463.295,A -85,B 0,C 180,E1 -1523.404,E2 -1523.404} C_VEL
LIN {X 0,Y 587.211,Z 469.682,A -85,B 0,C 180,E1 -1524.506,E2 -1524.506} C_VEL
LIN {X 0,Y 587.188,Z 474.377,A -85,B 0,C 180,E1 -1525.538,E2 -1525.538} C_VEL
LIN {X 0,Y 587.193,Z 477.964,A -85,B 0,C 180,E1 -1526.569,E2 -1526.569} C_VEL
LIN {X 0,Y 587.132,Z 479.796,A -85,B 0,C 180,E1 -1527.256,E2 -1527.256} C_VEL
LIN {X 0,Y 587.147,Z 482.188,A -85,B 0,C 180,E1 -1528.628,E2 -1528.628} C_VEL
LIN {X 0,Y 587.14,Z 482.782,A -85,B 0,C 180,E1 -1529.314,E2 -1529.314} C_VEL
LIN {X 0,Y 587.14,Z 482.782,A -85,B 0,C 180,E1 -1530.686,E2 -1530.686} C_VEL
LIN {X 0,Y 587.147,Z 482.188,A -85,B 0,C 180,E1 -1531.372,E2 -1531.372} C_VEL
LIN {X 0,Y 587.132,Z 479.796,A -85,B 0,C 180,E1 -1532.744,E2 -1532.744} C_VEL
LIN {X 0,Y 587.213,Z 476.884,A -85,B 0,C 180,E1 -1533.774,E2 -1533.774} C_VEL
LIN {X 0,Y 587.146,Z 472.935,A -85,B 0,C 180,E1 -1534.806,E2 -1534.806} C_VEL
LIN {X 0,Y 587.23,Z 467.84,A -85,B 0,C 180,E1 -1535.839,E2 -1535.839} C_VEL
LIN {X 0,Y 587.23,Z 461.457,A -85,B 0,C 180,E1 -1536.874,E2 -1536.874} C_VEL
LIN {X 0,Y 587.287,Z 453.488,A -85,B 0,C 180,E1 -1537.91,E2 -1537.91} C_VEL
LIN {X 0,Y 587.336,Z 445.347,A -85,B 0,C 180,E1 -1538.776,E2 -1538.776} C_VEL
LIN {X 0,Y 587.39,Z 435.362,A -85,B 0,C 180,E1 -1539.643,E2 -1539.643} C_VEL
LIN {X 0,Y 587.443,Z 425.544,A -85,B 0,C 180,E1 -1540.338,E2 -1540.338} C_VEL
LIN {X 0,Y 587.504,Z 414.935,A -85,B 0,C 180,E1 -1540.947,E2 -1540.947} C_VEL
LIN {X 0,Y 587.587,Z 401.419,A -85,B 0,C 180,E1 -1541.541,E2 -1541.541} C_VEL
LIN {X 0,Y 587.708,Z 388.986,A -85,B 0,C 180,E1 -1541.926,E2 -1541.926} C_VEL
LIN {X 0,Y 587.563,Z 380.116,A -85,B 0,C 180,E1 -1542.126,E2 -1542.126} C_VEL
LIN {X 0,Y 587.148,Z 377.523,A -85,B 0,C 180,E1 -1542.179,E2 -1542.179} C_VEL
LIN {X 0,Y 587.176,Z 371.46,A -85,B 0,C 180,E1 -1544.557,E2 -1544.557} C_VEL
LIN {X 0,Y 587.207,Z 364.274,A -85,B 0,C 180,E1 -1547.41,E2 -1547.41} C_VEL
LIN {X 0,Y 587.212,Z 358.884,A -85,B 0,C 180,E1 -1549.579,E2 -1549.579} C_VEL
LIN {X 0,Y 587.242,Z 353.495,A -85,B 0,C 180,E1 -1551.777,E2 -1551.777} C_VEL
LIN {X 0,Y 587.293,Z 346.309,A -85,B 0,C 180,E1 -1554.761,E2 -1554.761} C_VEL
LIN {X 0,Y 587.3,Z 339.495,A -85,B 0,C 180,E1 -1557.683,E2 -1557.683} C_VEL
LIN {X 0,Y 587.34,Z 333.889,A -85,B 0,C 180,E1 -1560.17,E2 -1560.17} C_VEL
LIN {X 0,Y 587.399,Z 327.661,A -85,B 0,C 180,E1 -1563.12,E2 -1563.12} C_VEL
LIN {X 0,Y 587.434,Z 322.777,A -85,B 0,C 180,E1 -1565.556,E2 -1565.556} C_VEL
LIN {X 0,Y 587.495,Z 318.406,A -85,B 0,C 180,E1 -1567.857,E2 -1567.857} C_VEL
LIN {X 0,Y 587.506,Z 314.149,A -85,B 0,C 180,E1 -1570.238,E2 -1570.238} C_VEL
LIN {X 0,Y 587.553,Z 310.968,A -85,B 0,C 180,E1 -1572.131,E2 -1572.131} C_VEL
LIN {X 0,Y 587.412,Z 309.371,A -85,B 0,C 180,E1 -1573.128,E2 -1573.128} C_VEL
LIN {X 0,Y 587.328,Z 308.829,A -85,B 0,C 180,E1 -1574.113,E2 -1574.113} C_VEL
LIN {X 0,Y 587.313,Z 308.823,A -85,B 0,C 180,E1 -1576.993,E2 -1576.993} C_VEL
LIN {X 0,Y 587.316,Z 308.825,A -85,B 0,C 180,E1 -1579.745,E2 -1579.745} C_VEL
LIN {X 0,Y 587.345,Z 308.823,A -85,B 0,C 180,E1 -1582.392,E2 -1582.392} C_VEL
LIN {X 0,Y 587.358,Z 308.822,A -85,B 0,C 180,E1 -1585.779,E2 -1585.779} C_VEL
LIN {X 0,Y 587.339,Z 308.823,A -85,B 0,C 180,E1 -1588.231,E2 -1588.231} C_VEL
LIN {X 0,Y 587.349,Z 308.816,A -85,B 0,C 180,E1 -1590.866,E2 -1590.866} C_VEL
LIN {X 0,Y 587.359,Z 308.826,A -85,B 0,C 180,E1 -1593.819,E2 -1593.819} C_VEL
LIN {X 0,Y 587.331,Z 308.825,A -85,B 0,C 180,E1 -1595.993,E2 -1595.993} C_VEL
LIN {X 0,Y 587.324,Z 308.822,A -85,B 0,C 180,E1 -1598.225,E2 -1598.225} C_VEL
LIN {X 0,Y 587.347,Z 308.82,A -85,B 0,C 180,E1 -1601.151,E2 -1601.151} C_VEL
LIN {X 0,Y 587.323,Z 308.823,A -85,B 0,C 180,E1 -1604.024,E2 -1604.024} C_VEL
LIN {X 0,Y 587.357,Z 308.817,A -85,B 0,C 180,E1 -1606.154,E2 -1606.154} C_VEL
LIN {X 0,Y 587.34,Z 308.82,A -85,B 0,C 180,E1 -1608.962,E2 -1608.962} C_VEL
LIN {X 0,Y 587.371,Z 308.818,A -85,B 0,C 180,E1 -1611.744,E2 -1611.744} C_VEL
LIN {X 0,Y 587.355,Z 308.816,A -85,B 0,C 180,E1 -1614.507,E2 -1614.507} C_VEL
LIN {X 0,Y 587.373,Z 308.824,A -85,B 0,C 180,E1 -1617.256,E2 -1617.256} C_VEL
LIN {X 0,Y 587.383,Z 308.813,A -85,B 0,C 180,E1 -1620,E2 -1620} C_VEL
LIN {X 0,Y 587.366,Z 308.819,A -85,B 0,C 180,E1 -1622.743,E2 -1622.743} C_VEL
LIN {X 0,Y 587.365,Z 308.818,A -85,B 0,C 180,E1 -1625.493,E2 -1625.493} C_VEL
LIN {X 0,Y 587.362,Z 308.816,A -85,B 0,C 180,E1 -1628.255,E2 -1628.255} C_VEL
LIN {X 0,Y 587.346,Z 308.823,A -85,B 0,C 180,E1 -1631.133,E2 -1631.133} C_VEL
LIN {X 0,Y 587.363,Z 308.817,A -85,B 0,C 180,E1 -1634.26,E2 -1634.26} C_VEL
LIN {X 0,Y 587.347,Z 308.818,A -85,B 0,C 180,E1 -1637.406,E2 -1637.406} C_VEL
LIN {X 0,Y 587.307,Z 308.824,A -85,B 0,C 180,E1 -1638.301,E2 -1638.301} C_VEL
LIN {X 0,Y 586.665,Z 308.909,A -85,B 0,C 180,E1 -1638.873,E2 -1638.873} C_VEL
LIN {X 0,Y 583.84,Z 309.261,A -85,B 0,C 180,E1 -1639.802,E2 -1639.802} C_VEL
LIN {X 0,Y 581.43,Z 309.562,A -85,B 0,C 180,E1 -1640.549,E2 -1640.549} C_VEL
LIN {X 0,Y 580.377,Z 309.688,A -85,B 0,C 180,E1 -1641.125,E2 -1641.125} C_VEL
LIN {X 0,Y 580.282,Z 309.698,A -85,B 0,C 180,E1 -1641.321,E2 -1641.321} C_VEL
LIN {X 0,Y 580.275,Z 309.698,A -85,B 0,C 180,E1 -1643.558,E2 -1643.558} C_VEL
LIN {X 0,Y 580.29,Z 309.697,A -85,B 0,C 180,E1 -1645.849,E2 -1645.849} C_VEL
LIN {X 0,Y 580.298,Z 309.7,A -85,B 0,C 180,E1 -1648.185,E2 -1648.185} C_VEL
LIN {X 0,Y 580.289,Z 309.702,A -85,B 0,C 180,E1 -1650.696,E2 -1650.696} C_VEL
LIN {X 0,Y 580.301,Z 309.695,A -85,B 0,C 180,E1 -1653.316,E2 -1653.316} C_VEL
LIN {X 0,Y 580.267,Z 309.701,A -85,B 0,C 180,E1 -1655.759,E2 -1655.759} C_VEL
LIN {X 0,Y 580.287,Z 309.705,A -85,B 0,C 180,E1 -1658.146,E2 -1658.146} C_VEL
LIN {X 0,Y 580.298,Z 309.696,A -85,B 0,C 180,E1 -1660.843,E2 -1660.843} C_VEL
LIN {X 0,Y 580.285,Z 309.699,A -85,B 0,C 180,E1 -1663.657,E2 -1663.657} C_VEL
LIN {X 0,Y 580.282,Z 309.699,A -85,B 0,C 180,E1 -1666.608,E2 -1666.608} C_VEL
LIN {X 0,Y 580.298,Z 309.695,A -85,B 0,C 180,E1 -1669.157,E2 -1669.157} C_VEL
LIN {X 0,Y 580.288,Z 309.706,A -85,B 0,C 180,E1 -1671.927,E2 -1671.927} C_VEL
LIN {X 0,Y 580.282,Z 309.699,A -85,B 0,C 180,E1 -1674.455,E2 -1674.455} C_VEL
LIN {X 0,Y 580.288,Z 309.696,A -85,B 0,C 180,E1 -1676.975,E2 -1676.975} C_VEL
LIN {X 0,Y 580.299,Z 309.7,A -85,B 0,C 180,E1 -1679.425,E2 -1679.425} C_VEL
LIN {X 0,Y 580.317,Z 309.696,A -85,B 0,C 180,E1 -1682.137,E2 -1682.137} C_VEL
LIN {X 0,Y 580.304,Z 309.695,A -85,B 0,C 180,E1 -1684.92,E2 -1684.92} C_VEL
LIN {X 0,Y 580.272,Z 309.702,A -85,B 0,C 180,E1 -1687.947,E2 -1687.947} C_VEL
LIN {X 0,Y 580.316,Z 309.695,A -85,B 0,C 180,E1 -1690.914,E2 -1690.914} C_VEL
LIN {X 0,Y 580.277,Z 309.702,A -85,B 0,C 180,E1 -1693.826,E2 -1693.826} C_VEL
LIN {X 0,Y 580.323,Z 309.694,A -85,B 0,C 180,E1 -1695.983,E2 -1695.983} C_VEL
LIN {X 0,Y 580.301,Z 309.698,A -85,B 0,C 180,E1 -1698.827,E2 -1698.827} C_VEL
LIN {X 0,Y 580.331,Z 309.695,A -85,B 0,C 180,E1 -1701.644,E2 -1701.644} C_VEL
LIN {X 0,Y 580.328,Z 309.693,A -85,B 0,C 180,E1 -1704.44,E2 -1704.44} C_VEL
LIN {X 0,Y 580.344,Z 309.69,A -85,B 0,C 180,E1 -1707.918,E2 -1707.918} C_VEL
LIN {X 0,Y 580.359,Z 309.693,A -85,B 0,C 180,E1 -1710.694,E2 -1710.694} C_VEL
LIN {X 0,Y 580.281,Z 309.7,A -85,B 0,C 180,E1 -1713.472,E2 -1713.472} C_VEL
LIN {X 0,Y 580.328,Z 309.693,A -85,B 0,C 180,E1 -1715.56,E2 -1715.56} C_VEL
LIN {X 0,Y 580.331,Z 309.695,A -85,B 0,C 180,E1 -1718.356,E2 -1718.356} C_VEL
LIN {X 0,Y 580.297,Z 309.699,A -85,B 0,C 180,E1 -1721.191,E2 -1721.191} C_VEL
LIN {X 0,Y 580.323,Z 309.694,A -85,B 0,C 180,E1 -1724.017,E2 -1724.017} C_VEL
LIN {X 0,Y 580.309,Z 309.699,A -85,B 0,C 180,E1 -1726.914,E2 -1726.914} C_VEL
LIN {X 0,Y 580.303,Z 309.695,A -85,B 0,C 180,E1 -1729.822,E2 -1729.822} C_VEL
LIN {X 0,Y 580.292,Z 309.7,A -85,B 0,C 180,E1 -1732.802,E2 -1732.802} C_VEL
LIN {X 0,Y 580.304,Z 309.695,A -85,B 0,C 180,E1 -1735.08,E2 -1735.08} C_VEL
LIN {X 0,Y 580.317,Z 309.696,A -85,B 0,C 180,E1 -1737.863,E2 -1737.863} C_VEL
LIN {X 0,Y 580.289,Z 309.699,A -85,B 0,C 180,E1 -1740.696,E2 -1740.696} C_VEL
LIN {X 0,Y 580.301,Z 309.695,A -85,B 0,C 180,E1 -1743.317,E2 -1743.317} C_VEL
LIN {X 0,Y 580.272,Z 309.702,A -85,B 0,C 180,E1 -1745.761,E2 -1745.761} C_VEL
LIN {X 0,Y 580.287,Z 309.705,A -85,B 0,C 180,E1 -1748.146,E2 -1748.146} C_VEL
LIN {X 0,Y 580.298,Z 309.695,A -85,B 0,C 180,E1 -1750.843,E2 -1750.843} C_VEL
LIN {X 0,Y 580.285,Z 309.702,A -85,B 0,C 180,E1 -1753.657,E2 -1753.657} C_VEL
LIN {X 0,Y 580.282,Z 309.698,A -85,B 0,C 180,E1 -1756.609,E2 -1756.609} C_VEL
LIN {X 0,Y 580.298,Z 309.696,A -85,B 0,C 180,E1 -1759.157,E2 -1759.157} C_VEL
LIN {X 0,Y 580.288,Z 309.703,A -85,B 0,C 180,E1 -1761.927,E2 -1761.927} C_VEL
LIN {X 0,Y 580.248,Z 309.702,A -85,B 0,C 180,E1 -1764.453,E2 -1764.453} C_VEL
LIN {X 0,Y 580.289,Z 309.697,A -85,B 0,C 180,E1 -1766.976,E2 -1766.976} C_VEL
LIN {X 0,Y 580.299,Z 309.703,A -85,B 0,C 180,E1 -1769.426,E2 -1769.426} C_VEL
LIN {X 0,Y 580.295,Z 309.696,A -85,B 0,C 180,E1 -1772.141,E2 -1772.141} C_VEL
LIN {X 0,Y 580.319,Z 309.7,A -85,B 0,C 180,E1 -1775.27,E2 -1775.27} C_VEL
LIN {X 0,Y 580.272,Z 309.7,A -85,B 0,C 180,E1 -1777.948,E2 -1777.948} C_VEL
LIN {X 0,Y 580.317,Z 309.697,A -85,B 0,C 180,E1 -1780.914,E2 -1780.914} C_VEL
LIN {X 0,Y 580.274,Z 309.699,A -85,B 0,C 180,E1 -1783.826,E2 -1783.826} C_VEL
LIN {X 0,Y 580.324,Z 309.692,A -85,B 0,C 180,E1 -1785.983,E2 -1785.983} C_VEL
LIN {X 0,Y 580.303,Z 309.7,A -85,B 0,C 180,E1 -1788.827,E2 -1788.827} C_VEL
LIN {X 0,Y 580.325,Z 309.693,A -85,B 0,C 180,E1 -1791.644,E2 -1791.644} C_VEL
LIN {X 0,Y 580.331,Z 309.693,A -85,B 0,C 180,E1 -1794.441,E2 -1794.441} C_VEL
LIN {X 0,Y 580.333,Z 309.695,A -85,B 0,C 180,E1 -1797.224,E2 -1797.224} C_VEL
LIN {X 0,Y 580.352,Z 309.688,A -85,B 0,C 180,E1 -1800,E2 -1800} C_VEL
LIN {X 0,Y 580.339,Z 309.7,A -85,B 0,C 180,E1 -1802.777,E2 -1802.777} C_VEL
LIN {X 0,Y 580.325,Z 309.692,A -85,B 0,C 180,E1 -1805.56,E2 -1805.56} C_VEL
LIN {X 0,Y 580.334,Z 309.696,A -85,B 0,C 180,E1 -1808.356,E2 -1808.356} C_VEL
LIN {X 0,Y 580.3,Z 309.696,A -85,B 0,C 180,E1 -1811.191,E2 -1811.191} C_VEL
LIN {X 0,Y 580.324,Z 309.695,A -85,B 0,C 180,E1 -1814.017,E2 -1814.017} C_VEL
LIN {X 0,Y 580.312,Z 309.696,A -85,B 0,C 180,E1 -1816.914,E2 -1816.914} C_VEL
LIN {X 0,Y 580.287,Z 309.699,A -85,B 0,C 180,E1 -1819.823,E2 -1819.823} C_VEL
LIN {X 0,Y 580.274,Z 309.704,A -85,B 0,C 180,E1 -1822.053,E2 -1822.053} C_VEL
LIN {X 0,Y 580.307,Z 309.694,A -85,B 0,C 180,E1 -1825.08,E2 -1825.08} C_VEL
LIN {X 0,Y 580.297,Z 309.704,A -85,B 0,C 180,E1 -1828.186,E2 -1828.186} C_VEL
LIN {X 0,Y 580.284,Z 309.698,A -85,B 0,C 180,E1 -1830.695,E2 -1830.695} C_VEL
LIN {X 0,Y 580.304,Z 309.695,A -85,B 0,C 180,E1 -1833.317,E2 -1833.317} C_VEL
LIN {X 0,Y 580.246,Z 309.708,A -85,B 0,C 180,E1 -1835.757,E2 -1835.757} C_VEL
LIN {X 0,Y 580.287,Z 309.703,A -85,B 0,C 180,E1 -1838.147,E2 -1838.147} C_VEL
LIN {X 0,Y 580.299,Z 309.696,A -85,B 0,C 180,E1 -1840.844,E2 -1840.844} C_VEL
LIN {X 0,Y 580.274,Z 309.708,A -85,B 0,C 180,E1 -1843.659,E2 -1843.659} C_VEL
LIN {X 0,Y 580.306,Z 309.844,A -85,B 0,C 180,E1 -1846.345,E2 -1846.345} C_VEL
LIN {X 0,Y 580.544,Z 312.834,A -85,B 0,C 180,E1 -1848.255,E2 -1848.255} C_VEL
LIN {X 0,Y 580.508,Z 317.5,A -85,B 0,C 180,E1 -1850.984,E2 -1850.984} C_VEL
LIN {X 0,Y 580.445,Z 322.291,A -85,B 0,C 180,E1 -1853.609,E2 -1853.609} C_VEL
LIN {X 0,Y 580.369,Z 327.234,A -85,B 0,C 180,E1 -1856.149,E2 -1856.149} C_VEL
LIN {X 0,Y 580.32,Z 332.291,A -85,B 0,C 180,E1 -1858.617,E2 -1858.617} C_VEL
LIN {X 0,Y 580.288,Z 337.483,A -85,B 0,C 180,E1 -1861.024,E2 -1861.024} C_VEL
LIN {X 0,Y 580.241,Z 343.468,A -85,B 0,C 180,E1 -1863.677,E2 -1863.677} C_VEL
LIN {X 0,Y 580.204,Z 348.105,A -85,B 0,C 180,E1 -1865.68,E2 -1865.68} C_VEL
LIN {X 0,Y 580.173,Z 355.291,A -85,B 0,C 180,E1 -1868.69,E2 -1868.69} C_VEL
LIN {X 0,Y 580.128,Z 362.478,A -85,B 0,C 180,E1 -1871.641,E2 -1871.641} C_VEL
LIN {X 0,Y 580.104,Z 369.664,A -85,B 0,C 180,E1 -1874.542,E2 -1874.542} C_VEL
LIN {X 0,Y 580.072,Z 375.053,A -85,B 0,C 180,E1 -1876.691,E2 -1876.691} C_VEL
LIN {X 0,Y 580.074,Z 377.523,A -85,B 0,C 180,E1 -1877.67,E2 -1877.67} C_VEL
LIN {X 0,Y 580.774,Z 383.531,A -85,B 0,C 180,E1 -1877.796,E2 -1877.796} C_VEL
LIN {X 0,Y 580.686,Z 395.811,A -85,B 0,C 180,E1 -1878.127,E2 -1878.127} C_VEL
LIN {X 0,Y 580.569,Z 407.706,A -85,B 0,C 180,E1 -1878.578,E2 -1878.578} C_VEL
LIN {X 0,Y 580.503,Z 419.769,A -85,B 0,C 180,E1 -1879.184,E2 -1879.184} C_VEL
LIN {X 0,Y 580.454,Z 430.748,A -85,B 0,C 180,E1 -1879.889,E2 -1879.889} C_VEL
LIN {X 0,Y 580.369,Z 439.637,A -85,B 0,C 180,E1 -1880.591,E2 -1880.591} C_VEL
LIN {X 0,Y 580.256,Z 448.758,A -85,B 0,C 180,E1 -1881.468,E2 -1881.468} C_VEL
LIN {X 0,Y 580.22,Z 456.305,A -85,B 0,C 180,E1 -1882.343,E2 -1882.343} C_VEL
LIN {X 0,Y 580.142,Z 463.793,A -85,B 0,C 180,E1 -1883.401,E2 -1883.401} C_VEL
LIN {X 0,Y 580.138,Z 469.682,A -85,B 0,C 180,E1 -1884.438,E2 -1884.438} C_VEL
LIN {X 0,Y 580.108,Z 474.379,A -85,B 0,C 180,E1 -1885.483,E2 -1885.483} C_VEL
LIN {X 0,Y 580.123,Z 477.966,A -85,B 0,C 180,E1 -1886.527,E2 -1886.527} C_VEL
LIN {X 0,Y 580.043,Z 479.791,A -85,B 0,C 180,E1 -1887.222,E2 -1887.222} C_VEL
LIN {X 0,Y 580.047,Z 482.19,A -85,B 0,C 180,E1 -1888.611,E2 -1888.611} C_VEL
LIN {X 0,Y 580.04,Z 482.782,A -85,B 0,C 180,E1 -1889.306,E2 -1889.306} C_VEL
LIN {X 0,Y 580.04,Z 482.782,A -85,B 0,C 180,E1 -1890.694,E2 -1890.694} C_VEL
LIN {X 0,Y 580.047,Z 482.19,A -85,B 0,C 180,E1 -1891.389,E2 -1891.389} C_VEL
LIN {X 0,Y 580.043,Z 479.791,A -85,B 0,C 180,E1 -1892.778,E2 -1892.778} C_VEL
LIN {X 0,Y 580.11,Z 476.878,A -85,B 0,C 180,E1 -1893.821,E2 -1893.821} C_VEL
LIN {X 0,Y 580.053,Z 472.927,A -85,B 0,C 180,E1 -1894.865,E2 -1894.865} C_VEL
LIN {X 0,Y 580.162,Z 467.832,A -85,B 0,C 180,E1 -1895.91,E2 -1895.91} C_VEL
LIN {X 0,Y 580.157,Z 461.448,A -85,B 0,C 180,E1 -1896.958,E2 -1896.958} C_VEL
LIN {X 0,Y 580.242,Z 453.491,A -85,B 0,C 180,E1 -1898.007,E2 -1898.007} C_VEL
LIN {X 0,Y 580.305,Z 445.35,A -85,B 0,C 180,E1 -1898.883,E2 -1898.883} C_VEL
LIN {X 0,Y 580.37,Z 435.35,A -85,B 0,C 180,E1 -1899.761,E2 -1899.761} C_VEL
LIN {X 0,Y 580.453,Z 425.529,A -85,B 0,C 180,E1 -1900.464,E2 -1900.464} C_VEL
LIN {X 0,Y 580.522,Z 414.93,A -85,B 0,C 180,E1 -1901.08,E2 -1901.08} C_VEL
LIN {X 0,Y 580.632,Z 402.154,A -85,B 0,C 180,E1 -1901.653,E2 -1901.653} C_VEL
LIN {X 0,Y 580.738,Z 389.83,A -85,B 0,C 180,E1 -1902.049,E2 -1902.049} C_VEL
LIN {X 0,Y 580.691,Z 381.269,A -85,B 0,C 180,E1 -1902.25,E2 -1902.25} C_VEL
LIN {X 0,Y 580.074,Z 377.523,A -85,B 0,C 180,E1 -1902.33,E2 -1902.33} C_VEL
LIN {X 0,Y 580.1,Z 371.46,A -85,B 0,C 180,E1 -1904.739,E2 -1904.739} C_VEL
LIN {X 0,Y 580.137,Z 364.274,A -85,B 0,C 180,E1 -1907.629,E2 -1907.629} C_VEL
LIN {X 0,Y 580.153,Z 358.884,A -85,B 0,C 180,E1 -1909.828,E2 -1909.828} C_VEL
LIN {X 0,Y 580.191,Z 353.495,A -85,B 0,C 180,E1 -1912.056,E2 -1912.056} C_VEL
LIN {X 0,Y 580.229,Z 346.317,A -85,B 0,C 180,E1 -1915.083,E2 -1915.083} C_VEL
LIN {X 0,Y 580.251,Z 340.009,A -85,B 0,C 180,E1 -1917.849,E2 -1917.849} C_VEL
LIN {X 0,Y 580.33,Z 333.714,A -85,B 0,C 180,E1 -1920.702,E2 -1920.702} C_VEL
LIN {X 0,Y 580.377,Z 328.268,A -85,B 0,C 180,E1 -1923.327,E2 -1923.327} C_VEL
LIN {X 0,Y 580.419,Z 323.449,A -85,B 0,C 180,E1 -1925.779,E2 -1925.779} C_VEL
LIN {X 0,Y 580.501,Z 319.057,A -85,B 0,C 180,E1 -1928.13,E2 -1928.13} C_VEL
LIN {X 0,Y 580.511,Z 314.364,A -85,B 0,C 180,E1 -1930.825,E2 -1930.825} C_VEL
LIN {X 0,Y 580.493,Z 311.325,A -85,B 0,C 180,E1 -1932.686,E2 -1932.686} C_VEL
LIN {X 0,Y 580.306,Z 309.835,A -85,B 0,C 180,E1 -1933.655,E2 -1933.655} C_VEL
LIN {X 0,Y 580.275,Z 309.704,A -85,B 0,C 180,E1 -1936.609,E2 -1936.609} C_VEL
LIN {X 0,Y 580.299,Z 309.696,A -85,B 0,C 180,E1 -1939.156,E2 -1939.156} C_VEL
LIN {X 0,Y 580.289,Z 309.704,A -85,B 0,C 180,E1 -1941.927,E2 -1941.927} C_VEL
LIN {X 0,Y 580.251,Z 309.705,A -85,B 0,C 180,E1 -1944.452,E2 -1944.452} C_VEL
LIN {X 0,Y 580.29,Z 309.696,A -85,B 0,C 180,E1 -1946.975,E2 -1946.975} C_VEL
LIN {X 0,Y 580.295,Z 309.698,A -85,B 0,C 180,E1 -1949.425,E2 -1949.425} C_VEL
LIN {X 0,Y 580.297,Z 309.7,A -85,B 0,C 180,E1 -1952.141,E2 -1952.141} C_VEL
LIN {X 0,Y 580.322,Z 309.694,A -85,B 0,C 180,E1 -1955.269,E2 -1955.269} C_VEL
LIN {X 0,Y 580.274,Z 309.704,A -85,B 0,C 180,E1 -1957.947,E2 -1957.947} C_VEL
LIN {X 0,Y 580.297,Z 309.696,A -85,B 0,C 180,E1 -1960.913,E2 -1960.913} C_VEL
LIN {X 0,Y 580.277,Z 309.703,A -85,B 0,C 180,E1 -1963.825,E2 -1963.825} C_VEL
LIN {X 0,Y 580.324,Z 309.695,A -85,B 0,C 180,E1 -1965.983,E2 -1965.983} C_VEL
LIN {X 0,Y 580.305,Z 309.695,A -85,B 0,C 180,E1 -1968.827,E2 -1968.827} C_VEL
LIN {X 0,Y 580.334,Z 309.696,A -85,B 0,C 180,E1 -1971.644,E2 -1971.644} C_VEL
LIN {X 0,Y 580.324,Z 309.692,A -85,B 0,C 180,E1 -1974.44,E2 -1974.44} C_VEL
LIN {X 0,Y 580.346,Z 309.69,A -85,B 0,C 180,E1 -1977.918,E2 -1977.918} C_VEL
LIN {X 0,Y 580.355,Z 309.691,A -85,B 0,C 180,E1 -1980.693,E2 -1980.693} C_VEL
LIN {X 0,Y 580.287,Z 309.7,A -85,B 0,C 180,E1 -1983.471,E2 -1983.471} C_VEL
LIN {X 0,Y 580.331,Z 309.693,A -85,B 0,C 180,E1 -1985.559,E2 -1985.559} C_VEL
LIN {X 0,Y 580.325,Z 309.693,A -85,B 0,C 180,E1 -1988.356,E2 -1988.356} C_VEL
LIN {X 0,Y 580.298,Z 309.7,A -85,B 0,C 180,E1 -1991.191,E2 -1991.191} C_VEL
LIN {X 0,Y 580.324,Z 309.692,A -85,B 0,C 180,E1 -1994.017,E2 -1994.017} C_VEL
LIN {X 0,Y 580.31,Z 309.701,A -85,B 0,C 180,E1 -1996.913,E2 -1996.913} C_VEL
LIN {X 0,Y 580.302,Z 309.694,A -85,B 0,C 180,E1 -1999.822,E2 -1999.822} C_VEL
LIN {X 0,Y 580.282,Z 309.698,A -85,B 0,C 180,E1 -2001.321,E2 -2001.321} C_VEL
LIN {X 0,Y 579.585,Z 309.785,A -85,B 0,C 180,E1 -2001.9,E2 -2001.9} C_VEL
LIN {X 0,Y 576.708,Z 310.149,A -85,B 0,C 180,E1 -2002.84,E2 -2002.84} C_VEL
LIN {X 0,Y 574.312,Z 310.443,A -85,B 0,C 180,E1 -2003.596,E2 -2003.596} C_VEL
LIN {X 0,Y 573.313,Z 310.569,A -85,B 0,C 180,E1 -2004.18,E2 -2004.18} C_VEL
LIN {X 0,Y 573.246,Z 310.578,A -85,B 0,C 180,E1 -2004.377,E2 -2004.377} C_VEL
LIN {X 0,Y 573.249,Z 310.576,A -85,B 0,C 180,E1 -2006.976,E2 -2006.976} C_VEL
LIN {X 0,Y 573.244,Z 310.574,A -85,B 0,C 180,E1 -2009.488,E2 -2009.488} C_VEL
LIN {X 0,Y 573.254,Z 310.579,A -85,B 0,C 180,E1 -2012.229,E2 -2012.229} C_VEL
LIN {X 0,Y 573.236,Z 310.578,A -85,B 0,C 180,E1 -2014.772,E2 -2014.772} C_VEL
LIN {X 0,Y 573.234,Z 310.578,A -85,B 0,C 180,E1 -2017.807,E2 -2017.807} C_VEL
LIN {X 0,Y 573.266,Z 310.575,A -85,B 0,C 180,E1 -2020.528,E2 -2020.528} C_VEL
LIN {X 0,Y 573.25,Z 310.576,A -85,B 0,C 180,E1 -2023.67,E2 -2023.67} C_VEL
LIN {X 0,Y 573.243,Z 310.575,A -85,B 0,C 180,E1 -2026.642,E2 -2026.642} C_VEL
LIN {X 0,Y 573.271,Z 310.573,A -85,B 0,C 180,E1 -2029.477,E2 -2029.477} C_VEL
LIN {X 0,Y 573.234,Z 310.58,A -85,B 0,C 180,E1 -2032.193,E2 -2032.193} C_VEL
LIN {X 0,Y 573.25,Z 310.573,A -85,B 0,C 180,E1 -2034.815,E2 -2034.815} C_VEL
LIN {X 0,Y 573.253,Z 310.576,A -85,B 0,C 180,E1 -2037.355,E2 -2037.355} C_VEL
LIN {X 0,Y 573.246,Z 310.582,A -85,B 0,C 180,E1 -2039.824,E2 -2039.824} C_VEL
LIN {X 0,Y 573.285,Z 310.57,A -85,B 0,C 180,E1 -2042.235,E2 -2042.235} C_VEL
LIN {X 0,Y 573.265,Z 310.574,A -85,B 0,C 180,E1 -2045.121,E2 -2045.121} C_VEL
LIN {X 0,Y 573.235,Z 310.583,A -85,B 0,C 180,E1 -2047.662,E2 -2047.662} C_VEL
LIN {X 0,Y 573.275,Z 310.57,A -85,B 0,C 180,E1 -2050.728,E2 -2050.728} C_VEL
LIN {X 0,Y 573.249,Z 310.58,A -85,B 0,C 180,E1 -2053.622,E2 -2053.622} C_VEL
LIN {X 0,Y 573.27,Z 310.574,A -85,B 0,C 180,E1 -2055.807,E2 -2055.807} C_VEL
LIN {X 0,Y 573.259,Z 310.575,A -85,B 0,C 180,E1 -2058.745,E2 -2058.745} C_VEL
LIN {X 0,Y 573.287,Z 310.574,A -85,B 0,C 180,E1 -2061.541,E2 -2061.541} C_VEL
LIN {X 0,Y 573.296,Z 310.569,A -85,B 0,C 180,E1 -2064.372,E2 -2064.372} C_VEL
LIN {X 0,Y 573.314,Z 310.566,A -85,B 0,C 180,E1 -2067.892,E2 -2067.892} C_VEL
LIN {X 0,Y 573.33,Z 310.569,A -85,B 0,C 180,E1 -2070.702,E2 -2070.702} C_VEL
LIN {X 0,Y 573.303,Z 310.575,A -85,B 0,C 180,E1 -2072.811,E2 -2072.811} C_VEL
LIN {X 0,Y 573.296,Z 310.569,A -85,B 0,C 180,E1 -2075.628,E2 -2075.628} C_VEL
LIN {X 0,Y 573.287,Z 310.574,A -85,B 0,C 180,E1 -2078.459,E2 -2078.459} C_VEL
LIN {X 0,Y 573.269,Z 310.573,A -85,B 0,C 180,E1 -2081.312,E2 -2081.312} C_VEL
LIN {X 0,Y 573.27,Z 310.574,A -85,B 0,C 180,E1 -2084.193,E2 -2084.193} C_VEL
LIN {X 0,Y 573.255,Z 310.575,A -85,B 0,C 180,E1 -2087.112,E2 -2087.112} C_VEL
LIN {X 0,Y 573.251,Z 310.576,A -85,B 0,C 180,E1 -2090.077,E2 -2090.077} C_VEL
LIN {X 0,Y 573.231,Z 310.576,A -85,B 0,C 180,E1 -2093.099,E2 -2093.099} C_VEL
LIN {X 0,Y 573.252,Z 310.573,A -85,B 0,C 180,E1 -2095.41,E2 -2095.41} C_VEL
LIN {X 0,Y 573.261,Z 310.577,A -85,B 0,C 180,E1 -2098.032,E2 -2098.032} C_VEL
LIN {X 0,Y 573.235,Z 310.576,A -85,B 0,C 180,E1 -2100.884,E2 -2100.884} C_VEL
LIN {X 0,Y 573.258,Z 310.573,A -85,B 0,C 180,E1 -2103.524,E2 -2103.524} C_VEL
LIN {X 0,Y 573.241,Z 310.583,A -85,B 0,C 180,E1 -2106.049,E2 -2106.049} C_VEL
LIN {X 0,Y 573.247,Z 310.575,A -85,B 0,C 180,E1 -2108.701,E2 -2108.701} C_VEL
LIN {X 0,Y 573.25,Z 310.577,A -85,B 0,C 180,E1 -2111.596,E2 -2111.596} C_VEL
LIN {X 0,Y 573.236,Z 310.578,A -85,B 0,C 180,E1 -2114.333,E2 -2114.333} C_VEL
LIN {X 0,Y 573.24,Z 310.577,A -85,B 0,C 180,E1 -2117.358,E2 -2117.358} C_VEL
LIN {X 0,Y 573.245,Z 310.575,A -85,B 0,C 180,E1 -2120.393,E2 -2120.393} C_VEL
LIN {X 0,Y 573.25,Z 310.574,A -85,B 0,C 180,E1 -2123.078,E2 -2123.078} C_VEL
LIN {X 0,Y 573.264,Z 310.581,A -85,B 0,C 180,E1 -2125.672,E2 -2125.672} C_VEL
LIN {X 0,Y 573.247,Z 310.575,A -85,B 0,C 180,E1 -2128.185,E2 -2128.185} C_VEL
LIN {X 0,Y 573.262,Z 310.571,A -85,B 0,C 180,E1 -2130.635,E2 -2130.635} C_VEL
LIN {X 0,Y 573.249,Z 310.576,A -85,B 0,C 180,E1 -2133.024,E2 -2133.024} C_VEL
LIN {X 0,Y 573.272,Z 310.579,A -85,B 0,C 180,E1 -2135.366,E2 -2135.366} C_VEL
LIN {X 0,Y 573.227,Z 310.576,A -85,B 0,C 180,E1 -2138.42,E2 -2138.42} C_VEL
LIN {X 0,Y 573.276,Z 310.572,A -85,B 0,C 180,E1 -2140.729,E2 -2140.729} C_VEL
LIN {X 0,Y 573.246,Z 310.577,A -85,B 0,C 180,E1 -2143.622,E2 -2143.622} C_VEL
LIN {X 0,Y 573.271,Z 310.571,A -85,B 0,C 180,E1 -2145.807,E2 -2145.807} C_VEL
LIN {X 0,Y 573.261,Z 310.576,A -85,B 0,C 180,E1 -2148.745,E2 -2148.745} C_VEL
LIN {X 0,Y 573.281,Z 310.571,A -85,B 0,C 180,E1 -2151.541,E2 -2151.541} C_VEL
LIN {X 0,Y 573.298,Z 310.569,A -85,B 0,C 180,E1 -2154.372,E2 -2154.372} C_VEL
LIN {X 0,Y 573.314,Z 310.565,A -85,B 0,C 180,E1 -2157.893,E2 -2157.893} C_VEL
LIN {X 0,Y 573.335,Z 310.571,A -85,B 0,C 180,E1 -2160.703,E2 -2160.703} C_VEL
LIN {X 0,Y 573.305,Z 310.575,A -85,B 0,C 180,E1 -2162.811,E2 -2162.811} C_VEL
LIN {X 0,Y 573.293,Z 310.567,A -85,B 0,C 180,E1 -2165.629,E2 -2165.629} C_VEL
LIN {X 0,Y 573.29,Z 310.575,A -85,B 0,C 180,E1 -2168.46,E2 -2168.46} C_VEL
LIN {X 0,Y 573.272,Z 310.571,A -85,B 0,C 180,E1 -2171.312,E2 -2171.312} C_VEL
LIN {X 0,Y 573.281,Z 310.578,A -85,B 0,C 180,E1 -2174.425,E2 -2174.425} C_VEL
LIN {X 0,Y 573.258,Z 310.573,A -85,B 0,C 180,E1 -2177.112,E2 -2177.112} C_VEL
LIN {X 0,Y 573.242,Z 310.58,A -85,B 0,C 180,E1 -2180.077,E2 -2180.077} C_VEL
LIN {X 0,Y 573.236,Z 310.584,A -85,B 0,C 180,E1 -2182.338,E2 -2182.338} C_VEL
LIN {X 0,Y 573.254,Z 310.573,A -85,B 0,C 180,E1 -2185.41,E2 -2185.41} C_VEL
LIN {X 0,Y 573.25,Z 310.581,A -85,B 0,C 180,E1 -2188.029,E2 -2188.029} C_VEL
LIN {X 0,Y 573.246,Z 310.582,A -85,B 0,C 180,E1 -2190.176,E2 -2190.176} C_VEL
LIN {X 0,Y 573.253,Z 310.574,A -85,B 0,C 180,E1 -2192.645,E2 -2192.645} C_VEL
LIN {X 0,Y 573.206,Z 310.579,A -85,B 0,C 180,E1 -2195.188,E2 -2195.188} C_VEL
LIN {X 0,Y 573.236,Z 310.584,A -85,B 0,C 180,E1 -2197.808,E2 -2197.808} C_VEL
LIN {X 0,Y 573.245,Z 310.576,A -85,B 0,C 180,E1 -2200.525,E2 -2200.525} C_VEL
LIN {X 0,Y 573.237,Z 310.58,A -85,B 0,C 180,E1 -2203.36,E2 -2203.36} C_VEL
LIN {X 0,Y 573.238,Z 310.584,A -85,B 0,C 180,E1 -2205.667,E2 -2205.667} C_VEL
LIN {X 0,Y 573.395,Z 311.577,A -85,B 0,C 180,E1 -2206.656,E2 -2206.656} C_VEL
LIN {X 0,Y 573.557,Z 314.587,A -85,B 0,C 180,E1 -2208.572,E2 -2208.572} C_VEL
LIN {X 0,Y 573.491,Z 319.257,A -85,B 0,C 180,E1 -2211.319,E2 -2211.319} C_VEL
LIN {X 0,Y 573.436,Z 324.116,A -85,B 0,C 180,E1 -2213.988,E2 -2213.988} C_VEL
LIN {X 0,Y 573.362,Z 329.035,A -85,B 0,C 180,E1 -2216.524,E2 -2216.524} C_VEL
LIN {X 0,Y 573.295,Z 334.293,A -85,B 0,C 180,E1 -2219.107,E2 -2219.107} C_VEL
LIN {X 0,Y 573.209,Z 339.314,A -85,B 0,C 180,E1 -2221.434,E2 -2221.434} C_VEL
LIN {X 0,Y 573.177,Z 344.591,A -85,B 0,C 180,E1 -2223.806,E2 -2223.806} C_VEL
LIN {X 0,Y 573.118,Z 349.876,A -85,B 0,C 180,E1 -2226.13,E2 -2226.13} C_VEL
LIN {X 0,Y 573.104,Z 357.088,A -85,B 0,C 180,E1 -2229.168,E2 -2229.168} C_VEL
LIN {X 0,Y 573.055,Z 362.478,A -85,B 0,C 180,E1 -2231.406,E2 -2231.406} C_VEL
LIN {X 0,Y 573.011,Z 369.664,A -85,B 0,C 180,E1 -2234.346,E2 -2234.346} C_VEL
LIN {X 0,Y 573.006,Z 375.053,A -85,B 0,C 180,E1 -2236.524,E2 -2236.524} C_VEL
LIN {X 0,Y 572.987,Z 377.523,A -85,B 0,C 180,E1 -2237.515,E2 -2237.515} C_VEL
LIN {X 0,Y 573.842,Z 383.531,A -85,B 0,C 180,E1 -2237.646,E2 -2237.646} C_VEL
LIN {X 0,Y 573.74,Z 395.796,A -85,B 0,C 180,E1 -2237.981,E2 -2237.981} C_VEL
LIN {X 0,Y 573.632,Z 407.441,A -85,B 0,C 180,E1 -2238.427,E2 -2238.427} C_VEL
LIN {X 0,Y 573.511,Z 418.469,A -85,B 0,C 180,E1 -2238.977,E2 -2238.977} C_VEL
LIN {X 0,Y 573.444,Z 429.486,A -85,B 0,C 180,E1 -2239.675,E2 -2239.675} C_VEL
LIN {X 0,Y 573.338,Z 439.633,A -85,B 0,C 180,E1 -2240.475,E2 -2240.475} C_VEL
LIN {X 0,Y 573.198,Z 448.751,A -85,B 0,C 180,E1 -2241.362,E2 -2241.362} C_VEL
LIN {X 0,Y 573.16,Z 456.298,A -85,B 0,C 180,E1 -2242.248,E2 -2242.248} C_VEL
LIN {X 0,Y 573.073,Z 463.65,A -85,B 0,C 180,E1 -2243.297,E2 -2243.297} C_VEL
LIN {X 0,Y 573.069,Z 469.683,A -85,B 0,C 180,E1 -2244.37,E2 -2244.37} C_VEL
LIN {X 0,Y 573.028,Z 474.381,A -85,B 0,C 180,E1 -2245.428,E2 -2245.428} C_VEL
LIN {X 0,Y 573.022,Z 477.969,A -85,B 0,C 180,E1 -2246.484,E2 -2246.484} C_VEL
LIN {X 0,Y 572.959,Z 479.787,A -85,B 0,C 180,E1 -2247.188,E2 -2247.188} C_VEL
LIN {X 0,Y 572.946,Z 482.191,A -85,B 0,C 180,E1 -2248.594,E2 -2248.594} C_VEL
LIN {X 0,Y 572.941,Z 482.781,A -85,B 0,C 180,E1 -2249.297,E2 -2249.297} C_VEL
LIN {X 0,Y 572.941,Z 482.781,A -85,B 0,C 180,E1 -2250.703,E2 -2250.703} C_VEL
LIN {X 0,Y 572.946,Z 482.191,A -85,B 0,C 180,E1 -2251.406,E2 -2251.406} C_VEL
LIN {X 0,Y 572.959,Z 479.787,A -85,B 0,C 180,E1 -2252.812,E2 -2252.812} C_VEL
LIN {X 0,Y 573.015,Z 476.871,A -85,B 0,C 180,E1 -2253.868,E2 -2253.868} C_VEL
LIN {X 0,Y 572.962,Z 472.92,A -85,B 0,C 180,E1 -2254.926,E2 -2254.926} C_VEL
LIN {X 0,Y 573.074,Z 467.824,A -85,B 0,C 180,E1 -2255.983,E2 -2255.983} C_VEL
LIN {X 0,Y 573.083,Z 461.44,A -85,B 0,C 180,E1 -2257.044,E2 -2257.044} C_VEL
LIN {X 0,Y 573.177,Z 453.494,A -85,B 0,C 180,E1 -2258.106,E2 -2258.106} C_VEL
LIN {X 0,Y 573.279,Z 445.353,A -85,B 0,C 180,E1 -2258.993,E2 -2258.993} C_VEL
LIN {X 0,Y 573.344,Z 435.339,A -85,B 0,C 180,E1 -2259.881,E2 -2259.881} C_VEL
LIN {X 0,Y 573.47,Z 425.515,A -85,B 0,C 180,E1 -2260.593,E2 -2260.593} C_VEL
LIN {X 0,Y 573.555,Z 414.745,A -85,B 0,C 180,E1 -2261.226,E2 -2261.226} C_VEL
LIN {X 0,Y 573.672,Z 402.16,A -85,B 0,C 180,E1 -2261.796,E2 -2261.796} C_VEL
LIN {X 0,Y 573.82,Z 389.8,A -85,B 0,C 180,E1 -2262.197,E2 -2262.197} C_VEL
LIN {X 0,Y 573.65,Z 381.564,A -85,B 0,C 180,E1 -2262.397,E2 -2262.397} C_VEL
LIN {X 0,Y 572.987,Z 377.523,A -85,B 0,C 180,E1 -2262.485,E2 -2262.485} C_VEL
LIN {X 0,Y 573.029,Z 371.46,A -85,B 0,C 180,E1 -2264.925,E2 -2264.925} C_VEL
LIN {X 0,Y 573.056,Z 364.274,A -85,B 0,C 180,E1 -2267.854,E2 -2267.854} C_VEL
LIN {X 0,Y 573.071,Z 358.884,A -85,B 0,C 180,E1 -2270.083,E2 -2270.083} C_VEL
LIN {X 0,Y 573.108,Z 353.495,A -85,B 0,C 180,E1 -2272.343,E2 -2272.343} C_VEL
LIN {X 0,Y 573.173,Z 347.603,A -85,B 0,C 180,E1 -2274.857,E2 -2274.857} C_VEL
LIN {X 0,Y 573.21,Z 341.08,A -85,B 0,C 180,E1 -2277.769,E2 -2277.769} C_VEL
LIN {X 0,Y 573.284,Z 335.793,A -85,B 0,C 180,E1 -2280.174,E2 -2280.174} C_VEL
LIN {X 0,Y 573.312,Z 330.685,A -85,B 0,C 180,E1 -2282.641,E2 -2282.641} C_VEL
LIN {X 0,Y 573.396,Z 325.685,A -85,B 0,C 180,E1 -2285.174,E2 -2285.174} C_VEL
LIN {X 0,Y 573.485,Z 320.826,A -85,B 0,C 180,E1 -2287.788,E2 -2287.788} C_VEL
LIN {X 0,Y 573.503,Z 316.022,A -85,B 0,C 180,E1 -2290.555,E2 -2290.555} C_VEL
LIN {X 0,Y 573.523,Z 312.605,A -85,B 0,C 180,E1 -2292.672,E2 -2292.672} C_VEL
LIN {X 0,Y 573.326,Z 311.078,A -85,B 0,C 180,E1 -2293.677,E2 -2293.677} C_VEL
LIN {X 0,Y 573.227,Z 310.583,A -85,B 0,C 180,E1 -2294.675,E2 -2294.675} C_VEL
LIN {X 0,Y 573.241,Z 310.578,A -85,B 0,C 180,E1 -2297.599,E2 -2297.599} C_VEL
LIN {X 0,Y 573.251,Z 310.577,A -85,B 0,C 180,E1 -2300.567,E2 -2300.567} C_VEL
LIN {X 0,Y 573.253,Z 310.574,A -85,B 0,C 180,E1 -2303.077,E2 -2303.077} C_VEL
LIN {X 0,Y 573.266,Z 310.577,A -85,B 0,C 180,E1 -2305.671,E2 -2305.671} C_VEL
LIN {X 0,Y 573.239,Z 310.58,A -85,B 0,C 180,E1 -2308.184,E2 -2308.184} C_VEL
LIN {X 0,Y 573.264,Z 310.572,A -85,B 0,C 180,E1 -2310.634,E2 -2310.634} C_VEL
LIN {X 0,Y 573.25,Z 310.573,A -85,B 0,C 180,E1 -2313.024,E2 -2313.024} C_VEL
LIN {X 0,Y 573.275,Z 310.573,A -85,B 0,C 180,E1 -2315.366,E2 -2315.366} C_VEL
LIN {X 0,Y 573.23,Z 310.576,A -85,B 0,C 180,E1 -2318.419,E2 -2318.419} C_VEL
LIN {X 0,Y 573.269,Z 310.571,A -85,B 0,C 180,E1 -2320.731,E2 -2320.731} C_VEL
LIN {X 0,Y 573.249,Z 310.582,A -85,B 0,C 180,E1 -2323.621,E2 -2323.621} C_VEL
LIN {X 0,Y 573.272,Z 310.575,A -85,B 0,C 180,E1 -2325.807,E2 -2325.807} C_VEL
LIN {X 0,Y 573.263,Z 310.572,A -85,B 0,C 180,E1 -2328.745,E2 -2328.745} C_VEL
LIN {X 0,Y 573.29,Z 310.575,A -85,B 0,C 180,E1 -2331.54,E2 -2331.54} C_VEL
LIN {X 0,Y 573.293,Z 310.568,A -85,B 0,C 180,E1 -2334.371,E2 -2334.371} C_VEL
LIN {X 0,Y 573.316,Z 310.566,A -85,B 0,C 180,E1 -2337.892,E2 -2337.892} C_VEL
LIN {X 0,Y 573.326,Z 310.566,A -85,B 0,C 180,E1 -2340.702,E2 -2340.702} C_VEL
LIN {X 0,Y 573.301,Z 310.572,A -85,B 0,C 180,E1 -2342.81,E2 -2342.81} C_VEL
LIN {X 0,Y 573.298,Z 310.569,A -85,B 0,C 180,E1 -2345.628,E2 -2345.628} C_VEL
LIN {X 0,Y 573.281,Z 310.571,A -85,B 0,C 180,E1 -2348.459,E2 -2348.459} C_VEL
LIN {X 0,Y 573.27,Z 310.574,A -85,B 0,C 180,E1 -2351.312,E2 -2351.312} C_VEL
LIN {X 0,Y 573.28,Z 310.573,A -85,B 0,C 180,E1 -2354.424,E2 -2354.424} C_VEL
LIN {X 0,Y 573.256,Z 310.576,A -85,B 0,C 180,E1 -2357.111,E2 -2357.111} C_VEL
LIN {X 0,Y 573.25,Z 310.574,A -85,B 0,C 180,E1 -2360.076,E2 -2360.076} C_VEL
LIN {X 0,Y 573.232,Z 310.578,A -85,B 0,C 180,E1 -2363.099,E2 -2363.099} C_VEL
LIN {X 0,Y 573.246,Z 310.578,A -85,B 0,C 180,E1 -2364.377,E2 -2364.377} C_VEL
LIN {X 0,Y 572.62,Z 310.662,A -85,B 0,C 180,E1 -2364.964,E2 -2364.964} C_VEL
LIN {X 0,Y 569.779,Z 311.014,A -85,B 0,C 180,E1 -2365.915,E2 -2365.915} C_VEL
LIN {X 0,Y 567.348,Z 311.316,A -85,B 0,C 180,E1 -2366.681,E2 -2366.681} C_VEL
LIN {X 0,Y 566.292,Z 311.441,A -85,B 0,C 180,E1 -2367.272,E2 -2367.272} C_VEL
LIN {X 0,Y 566.201,Z 311.451,A -85,B 0,C 180,E1 -2367.472,E2 -2367.472} C_VEL
LIN {X 0,Y 566.199,Z 311.452,A -85,B 0,C 180,E1 -2369.768,E2 -2369.768} C_VEL
LIN {X 0,Y 566.206,Z 311.46,A -85,B 0,C 180,E1 -2372.431,E2 -2372.431} C_VEL
LIN {X 0,Y 566.197,Z 311.453,A -85,B 0,C 180,E1 -2374.992,E2 -2374.992} C_VEL
LIN {X 0,Y 566.194,Z 311.452,A -85,B 0,C 180,E1 -2377.46,E2 -2377.46} C_VEL
LIN {X 0,Y 566.224,Z 311.458,A -85,B 0,C 180,E1 -2380.197,E2 -2380.197} C_VEL
LIN {X 0,Y 566.202,Z 311.451,A -85,B 0,C 180,E1 -2383.053,E2 -2383.053} C_VEL
LIN {X 0,Y 566.199,Z 311.461,A -85,B 0,C 180,E1 -2386.048,E2 -2386.048} C_VEL
LIN {X 0,Y 566.209,Z 311.45,A -85,B 0,C 180,E1 -2388.864,E2 -2388.864} C_VEL
LIN {X 0,Y 566.187,Z 311.458,A -85,B 0,C 180,E1 -2391.637,E2 -2391.637} C_VEL
LIN {X 0,Y 566.192,Z 311.455,A -85,B 0,C 180,E1 -2394.31,E2 -2394.31} C_VEL
LIN {X 0,Y 566.226,Z 311.448,A -85,B 0,C 180,E1 -2396.898,E2 -2396.898} C_VEL
LIN {X 0,Y 566.185,Z 311.458,A -85,B 0,C 180,E1 -2399.408,E2 -2399.408} C_VEL
LIN {X 0,Y 566.225,Z 311.455,A -85,B 0,C 180,E1 -2401.858,E2 -2401.858} C_VEL
LIN {X 0,Y 566.221,Z 311.45,A -85,B 0,C 180,E1 -2404.252,E2 -2404.252} C_VEL
LIN {X 0,Y 566.17,Z 311.455,A -85,B 0,C 180,E1 -2406.718,E2 -2406.718} C_VEL
LIN {X 0,Y 566.212,Z 311.457,A -85,B 0,C 180,E1 -2409.663,E2 -2409.663} C_VEL
LIN {X 0,Y 566.197,Z 311.453,A -85,B 0,C 180,E1 -2412.668,E2 -2412.668} C_VEL
LIN {X 0,Y 566.231,Z 311.454,A -85,B 0,C 180,E1 -2415.627,E2 -2415.627} C_VEL
LIN {X 0,Y 566.232,Z 311.449,A -85,B 0,C 180,E1 -2418.675,E2 -2418.675} C_VEL
LIN {X 0,Y 566.231,Z 311.454,A -85,B 0,C 180,E1 -2421.434,E2 -2421.434} C_VEL
LIN {X 0,Y 566.265,Z 311.444,A -85,B 0,C 180,E1 -2424.302,E2 -2424.302} C_VEL
LIN {X 0,Y 566.284,Z 311.442,A -85,B 0,C 180,E1 -2427.866,E2 -2427.866} C_VEL
LIN {X 0,Y 566.3,Z 311.445,A -85,B 0,C 180,E1 -2430.711,E2 -2430.711} C_VEL
LIN {X 0,Y 566.269,Z 311.452,A -85,B 0,C 180,E1 -2432.846,E2 -2432.846} C_VEL
LIN {X 0,Y 566.265,Z 311.444,A -85,B 0,C 180,E1 -2435.698,E2 -2435.698} C_VEL
LIN {X 0,Y 566.231,Z 311.454,A -85,B 0,C 180,E1 -2438.566,E2 -2438.566} C_VEL
LIN {X 0,Y 566.239,Z 311.448,A -85,B 0,C 180,E1 -2441.454,E2 -2441.454} C_VEL
LIN {X 0,Y 566.231,Z 311.456,A -85,B 0,C 180,E1 -2444.507,E2 -2444.507} C_VEL
LIN {X 0,Y 566.197,Z 311.453,A -85,B 0,C 180,E1 -2447.332,E2 -2447.332} C_VEL
LIN {X 0,Y 566.212,Z 311.457,A -85,B 0,C 180,E1 -2450.337,E2 -2450.337} C_VEL
LIN {X 0,Y 566.17,Z 311.455,A -85,B 0,C 180,E1 -2453.282,E2 -2453.282} C_VEL
LIN {X 0,Y 566.221,Z 311.45,A -85,B 0,C 180,E1 -2455.748,E2 -2455.748} C_VEL
LIN {X 0,Y 566.203,Z 311.459,A -85,B 0,C 180,E1 -2458.203,E2 -2458.203} C_VEL
LIN {X 0,Y 566.196,Z 311.452,A -85,B 0,C 180,E1 -2461.078,E2 -2461.078} C_VEL
LIN {X 0,Y 566.208,Z 311.453,A -85,B 0,C 180,E1 -2463.734,E2 -2463.734} C_VEL
LIN {X 0,Y 566.208,Z 311.453,A -85,B 0,C 180,E1 -2466.569,E2 -2466.569} C_VEL
LIN {X 0,Y 566.21,Z 311.454,A -85,B 0,C 180,E1 -2469.686,E2 -2469.686} C_VEL
LIN {X 0,Y 566.211,Z 311.458,A -85,B 0,C 180,E1 -2472.087,E2 -2472.087} C_VEL
LIN {X 0,Y 566.171,Z 311.455,A -85,B 0,C 180,E1 -2475.036,E2 -2475.036} C_VEL
LIN {X 0,Y 566.215,Z 311.454,A -85,B 0,C 180,E1 -2478.136,E2 -2478.136} C_VEL
LIN {X 0,Y 566.219,Z 311.449,A -85,B 0,C 180,E1 -2480.727,E2 -2480.727} C_VEL
LIN {X 0,Y 566.181,Z 311.462,A -85,B 0,C 180,E1 -2483.788,E2 -2483.788} C_VEL
LIN {X 0,Y 566.208,Z 311.451,A -85,B 0,C 180,E1 -2486.266,E2 -2486.266} C_VEL
LIN {X 0,Y 566.196,Z 311.453,A -85,B 0,C 180,E1 -2488.922,E2 -2488.922} C_VEL
LIN {X 0,Y 566.209,Z 311.454,A -85,B 0,C 180,E1 -2491.858,E2 -2491.858} C_VEL
LIN {X 0,Y 566.211,Z 311.45,A -85,B 0,C 180,E1 -2494.251,E2 -2494.251} C_VEL
LIN {X 0,Y 566.17,Z 311.456,A -85,B 0,C 180,E1 -2496.719,E2 -2496.719} C_VEL
LIN {X 0,Y 566.211,Z 311.454,A -85,B 0,C 180,E1 -2499.663,E2 -2499.663} C_VEL
LIN {X 0,Y 566.197,Z 311.453,A -85,B 0,C 180,E1 -2502.669,E2 -2502.669} C_VEL
LIN {X 0,Y 566.232,Z 311.45,A -85,B 0,C 180,E1 -2505.627,E2 -2505.627} C_VEL
LIN {X 0,Y 566.233,Z 311.45,A -85,B 0,C 180,E1 -2508.676,E2 -2508.676} C_VEL
LIN {X 0,Y 566.226,Z 311.452,A -85,B 0,C 180,E1 -2511.435,E2 -2511.435} C_VEL
LIN {X 0,Y 566.266,Z 311.444,A -85,B 0,C 180,E1 -2514.302,E2 -2514.302} C_VEL
LIN {X 0,Y 566.284,Z 311.441,A -85,B 0,C 180,E1 -2517.867,E2 -2517.867} C_VEL
LIN {X 0,Y 566.305,Z 311.446,A -85,B 0,C 180,E1 -2520.711,E2 -2520.711} C_VEL
LIN {X 0,Y 566.271,Z 311.451,A -85,B 0,C 180,E1 -2522.846,E2 -2522.846} C_VEL
LIN {X 0,Y 566.262,Z 311.443,A -85,B 0,C 180,E1 -2525.699,E2 -2525.699} C_VEL
LIN {X 0,Y 566.233,Z 311.456,A -85,B 0,C 180,E1 -2528.566,E2 -2528.566} C_VEL
LIN {X 0,Y 566.241,Z 311.446,A -85,B 0,C 180,E1 -2531.455,E2 -2531.455} C_VEL
LIN {X 0,Y 566.234,Z 311.456,A -85,B 0,C 180,E1 -2534.507,E2 -2534.507} C_VEL
LIN {X 0,Y 566.198,Z 311.451,A -85,B 0,C 180,E1 -2537.332,E2 -2537.332} C_VEL
LIN {X 0,Y 566.208,Z 311.46,A -85,B 0,C 180,E1 -2540.338,E2 -2540.338} C_VEL
LIN {X 0,Y 566.169,Z 311.455,A -85,B 0,C 180,E1 -2543.281,E2 -2543.281} C_VEL
LIN {X 0,Y 566.214,Z 311.452,A -85,B 0,C 180,E1 -2545.749,E2 -2545.749} C_VEL
LIN {X 0,Y 566.203,Z 311.46,A -85,B 0,C 180,E1 -2548.202,E2 -2548.202} C_VEL
LIN {X 0,Y 566.19,Z 311.452,A -85,B 0,C 180,E1 -2551.077,E2 -2551.077} C_VEL
LIN {X 0,Y 566.212,Z 311.455,A -85,B 0,C 180,E1 -2553.734,E2 -2553.734} C_VEL
LIN {X 0,Y 566.2,Z 311.454,A -85,B 0,C 180,E1 -2556.57,E2 -2556.57} C_VEL
LIN {X 0,Y 566.222,Z 311.457,A -85,B 0,C 180,E1 -2559.687,E2 -2559.687} C_VEL
LIN {X 0,Y 566.202,Z 311.454,A -85,B 0,C 180,E1 -2562.917,E2 -2562.917} C_VEL
LIN {X 0,Y 566.174,Z 311.46,A -85,B 0,C 180,E1 -2565.036,E2 -2565.036} C_VEL
LIN {X 0,Y 566.286,Z 311.92,A -85,B 0,C 180,E1 -2566.04,E2 -2566.04} C_VEL
LIN {X 0,Y 566.545,Z 315.049,A -85,B 0,C 180,E1 -2568.1,E2 -2568.1} C_VEL
LIN {X 0,Y 566.512,Z 319.443,A -85,B 0,C 180,E1 -2570.751,E2 -2570.751} C_VEL
LIN {X 0,Y 566.44,Z 324.214,A -85,B 0,C 180,E1 -2573.448,E2 -2573.448} C_VEL
LIN {X 0,Y 566.346,Z 329.518,A -85,B 0,C 180,E1 -2576.246,E2 -2576.246} C_VEL
LIN {X 0,Y 566.252,Z 334.865,A -85,B 0,C 180,E1 -2578.914,E2 -2578.914} C_VEL
LIN {X 0,Y 566.176,Z 339.326,A -85,B 0,C 180,E1 -2581.046,E2 -2581.046} C_VEL
LIN {X 0,Y 566.118,Z 344.588,A -85,B 0,C 180,E1 -2583.454,E2 -2583.454} C_VEL
LIN {X 0,Y 566.076,Z 349.849,A -85,B 0,C 180,E1 -2585.814,E2 -2585.814} C_VEL
LIN {X 0,Y 566.041,Z 357.088,A -85,B 0,C 180,E1 -2588.896,E2 -2588.896} C_VEL
LIN {X 0,Y 566.006,Z 362.478,A -85,B 0,C 180,E1 -2591.165,E2 -2591.165} C_VEL
LIN {X 0,Y 565.924,Z 369.664,A -85,B 0,C 180,E1 -2594.145,E2 -2594.145} C_VEL
LIN {X 0,Y 565.929,Z 375.053,A -85,B 0,C 180,E1 -2596.352,E2 -2596.352} C_VEL
LIN {X 0,Y 565.897,Z 377.523,A -85,B 0,C 180,E1 -2597.356,E2 -2597.356} C_VEL
LIN {X 0,Y 566.895,Z 384.47,A -85,B 0,C 180,E1 -2597.515,E2 -2597.515} C_VEL
LIN {X 0,Y 566.769,Z 397.072,A -85,B 0,C 180,E1 -2597.876,E2 -2597.876} C_VEL
LIN {X 0,Y 566.665,Z 408.429,A -85,B 0,C 180,E1 -2598.328,E2 -2598.328} C_VEL
LIN {X 0,Y 566.522,Z 420.349,A -85,B 0,C 180,E1 -2598.947,E2 -2598.947} C_VEL
LIN {X 0,Y 566.44,Z 431.914,A -85,B 0,C 180,E1 -2599.726,E2 -2599.726} C_VEL
LIN {X 0,Y 566.304,Z 441.559,A -85,B 0,C 180,E1 -2600.536,E2 -2600.536} C_VEL
LIN {X 0,Y 566.166,Z 450.365,A -85,B 0,C 180,E1 -2601.433,E2 -2601.433} C_VEL
LIN {X 0,Y 566.056,Z 459.008,A -85,B 0,C 180,E1 -2602.509,E2 -2602.509} C_VEL
LIN {X 0,Y 565.965,Z 465.875,A -85,B 0,C 180,E1 -2603.583,E2 -2603.583} C_VEL
LIN {X 0,Y 565.937,Z 471.363,A -85,B 0,C 180,E1 -2604.656,E2 -2604.656} C_VEL
LIN {X 0,Y 565.959,Z 475.657,A -85,B 0,C 180,E1 -2605.727,E2 -2605.727} C_VEL
LIN {X 0,Y 565.927,Z 477.971,A -85,B 0,C 180,E1 -2606.44,E2 -2606.44} C_VEL
LIN {X 0,Y 565.878,Z 479.782,A -85,B 0,C 180,E1 -2607.152,E2 -2607.152} C_VEL
LIN {X 0,Y 565.846,Z 482.193,A -85,B 0,C 180,E1 -2608.577,E2 -2608.577} C_VEL
LIN {X 0,Y 565.841,Z 482.781,A -85,B 0,C 180,E1 -2609.288,E2 -2609.288} C_VEL
LIN {X 0,Y 565.841,Z 482.781,A -85,B 0,C 180,E1 -2610.712,E2 -2610.712} C_VEL
LIN {X 0,Y 565.846,Z 482.193,A -85,B 0,C 180,E1 -2611.423,E2 -2611.423} C_VEL
LIN {X 0,Y 565.878,Z 479.782,A -85,B 0,C 180,E1 -2612.848,E2 -2612.848} C_VEL
LIN {X 0,Y 565.926,Z 476.865,A -85,B 0,C 180,E1 -2613.916,E2 -2613.916} C_VEL
LIN {X 0,Y 565.877,Z 472.912,A -85,B 0,C 180,E1 -2614.987,E2 -2614.987} C_VEL
LIN {X 0,Y 565.99,Z 467.815,A -85,B 0,C 180,E1 -2616.059,E2 -2616.059} C_VEL
LIN {X 0,Y 566.032,Z 461.432,A -85,B 0,C 180,E1 -2617.132,E2 -2617.132} C_VEL
LIN {X 0,Y 566.131,Z 453.497,A -85,B 0,C 180,E1 -2618.208,E2 -2618.208} C_VEL
LIN {X 0,Y 566.238,Z 445.356,A -85,B 0,C 180,E1 -2619.105,E2 -2619.105} C_VEL
LIN {X 0,Y 566.343,Z 435.327,A -85,B 0,C 180,E1 -2620.005,E2 -2620.005} C_VEL
LIN {X 0,Y 566.486,Z 425.501,A -85,B 0,C 180,E1 -2620.725,E2 -2620.725} C_VEL
LIN {X 0,Y 566.563,Z 414.73,A -85,B 0,C 180,E1 -2621.367,E2 -2621.367} C_VEL
LIN {X 0,Y 566.717,Z 400.935,A -85,B 0,C 180,E1 -2621.989,E2 -2621.989} C_VEL
LIN {X 0,Y 566.888,Z 388.897,A -85,B 0,C 180,E1 -2622.371,E2 -2622.371} C_VEL
LIN {X 0,Y 566.624,Z 381.857,A -85,B 0,C 180,E1 -2622.548,E2 -2622.548} C_VEL
LIN {X 0,Y 565.897,Z 377.523,A -85,B 0,C 180,E1 -2622.644,E2 -2622.644} C_VEL
LIN {X 0,Y 565.939,Z 371.46,A -85,B 0,C 180,E1 -2625.117,E2 -2625.117} C_VEL
LIN {X 0,Y 565.984,Z 364.274,A -85,B 0,C 180,E1 -2628.085,E2 -2628.085} C_VEL
LIN {X 0,Y 566.007,Z 358.884,A -85,B 0,C 180,E1 -2630.345,E2 -2630.345} C_VEL
LIN {X 0,Y 566.053,Z 351.987,A -85,B 0,C 180,E1 -2633.253,E2 -2633.253} C_VEL
LIN {X 0,Y 566.109,Z 346.342,A -85,B 0,C 180,E1 -2635.754,E2 -2635.754} C_VEL
LIN {X 0,Y 566.151,Z 340.981,A -85,B 0,C 180,E1 -2638.191,E2 -2638.191} C_VEL
LIN {X 0,Y 566.24,Z 335.869,A -85,B 0,C 180,E1 -2640.589,E2 -2640.589} C_VEL
LIN {X 0,Y 566.312,Z 330.778,A -85,B 0,C 180,E1 -2643.096,E2 -2643.096} C_VEL
LIN {X 0,Y 566.39,Z 325.832,A -85,B 0,C 180,E1 -2645.675,E2 -2645.675} C_VEL
LIN {X 0,Y 566.477,Z 320.981,A -85,B 0,C 180,E1 -2648.34,E2 -2648.34} C_VEL
